LIN {X 0,Y 310.585,Z 527.407,A -85,B 0,C 180,E1 -15760.43,E2 -15760.43} C_VEL
LIN {X 0,Y 310.715,Z 527.488,A -85,B 0,C 180,E1 -15761.746,E2 -15761.746} C_VEL
LIN {X 0,Y 310.944,Z 526.948,A -85,B 0,C 180,E1 -15763.618,E2 -15763.618} C_VEL
LIN {X 0,Y 311.218,Z 525.347,A -85,B 0,C 180,E1 -15765.723,E2 -15765.723} C_VEL
LIN {X 0,Y 311.749,Z 522.836,A -85,B 0,C 180,E1 -15767.719,E2 -15767.719} C_VEL
LIN {X 0,Y 312.493,Z 519.275,A -85,B 0,C 180,E1 -15769.716,E2 -15769.716} C_VEL
LIN {X 0,Y 313.497,Z 514.55,A -85,B 0,C 180,E1 -15771.71,E2 -15771.71} C_VEL
LIN {X 0,Y 314.758,Z 508.405,A -85,B 0,C 180,E1 -15773.73,E2 -15773.73} C_VEL
LIN {X 0,Y 316.283,Z 500.927,A -85,B 0,C 180,E1 -15775.678,E2 -15775.678} C_VEL
LIN {X 0,Y 317.858,Z 493.142,A -85,B 0,C 180,E1 -15777.309,E2 -15777.309} C_VEL
LIN {X 0,Y 319.637,Z 483.592,A -85,B 0,C 180,E1 -15778.929,E2 -15778.929} C_VEL
LIN {X 0,Y 321.405,Z 472.884,A -85,B 0,C 180,E1 -15780.376,E2 -15780.376} C_VEL
LIN {X 0,Y 322.865,Z 462.517,A -85,B 0,C 180,E1 -15781.495,E2 -15781.495} C_VEL
LIN {X 0,Y 324.159,Z 451.225,A -85,B 0,C 180,E1 -15782.457,E2 -15782.457} C_VEL
LIN {X 0,Y 325.243,Z 438.611,A -85,B 0,C 180,E1 -15783.252,E2 -15783.252} C_VEL
LIN {X 0,Y 325.852,Z 426.556,A -85,B 0,C 180,E1 -15783.783,E2 -15783.783} C_VEL
LIN {X 0,Y 326.612,Z 407.281,A -85,B 0,C 180,E1 -15784.25,E2 -15784.25} C_VEL
LIN {X 0,Y 328.373,Z 349.267,A -85,B 0,C 180,E1 -15785.509,E2 -15785.509} C_VEL
LIN {X 0,Y 326.303,Z 343.527,A -85,B 0,C 180,E1 -15785.856,E2 -15785.856} C_VEL
LIN {X 0,Y 318.976,Z 327.276,A -85,B 0,C 180,E1 -15787.031,E2 -15787.031} C_VEL
LIN {X 0,Y 315.882,Z 321.035,A -85,B 0,C 180,E1 -15787.532,E2 -15787.532} C_VEL
LIN {X 0,Y 314.268,Z 318.796,A -85,B 0,C 180,E1 -15787.811,E2 -15787.811} C_VEL
LIN {X 0,Y 311.353,Z 316.882,A -85,B 0,C 180,E1 -15788.356,E2 -15788.356} C_VEL
LIN {X 0,Y 308.133,Z 315.361,A -85,B 0,C 180,E1 -15789.123,E2 -15789.123} C_VEL
LIN {X 0,Y 306.033,Z 313.784,A -85,B 0,C 180,E1 -15789.924,E2 -15789.924} C_VEL
LIN {X 0,Y 305.457,Z 312.436,A -85,B 0,C 180,E1 -15790.569,E2 -15790.569} C_VEL
LIN {X 0,Y 305.425,Z 312.439,A -85,B 0,C 180,E1 -15793.655,E2 -15793.655} C_VEL
LIN {X 0,Y 305.454,Z 312.435,A -85,B 0,C 180,E1 -15797.414,E2 -15797.414} C_VEL
LIN {X 0,Y 305.467,Z 312.429,A -85,B 0,C 180,E1 -15801.596,E2 -15801.596} C_VEL
LIN {X 0,Y 305.462,Z 312.43,A -85,B 0,C 180,E1 -15804.887,E2 -15804.887} C_VEL
LIN {X 0,Y 305.451,Z 312.427,A -85,B 0,C 180,E1 -15808.355,E2 -15808.355} C_VEL
LIN {X 0,Y 305.52,Z 312.423,A -85,B 0,C 180,E1 -15811.114,E2 -15811.114} C_VEL
LIN {X 0,Y 305.571,Z 312.415,A -85,B 0,C 180,E1 -15814.088,E2 -15814.088} C_VEL
LIN {X 0,Y 305.482,Z 312.428,A -85,B 0,C 180,E1 -15818.402,E2 -15818.402} C_VEL
LIN {X 0,Y 305.58,Z 312.412,A -85,B 0,C 180,E1 -15821.217,E2 -15821.217} C_VEL
LIN {X 0,Y 305.649,Z 312.404,A -85,B 0,C 180,E1 -15825.349,E2 -15825.349} C_VEL
LIN {X 0,Y 305.639,Z 312.405,A -85,B 0,C 180,E1 -15829.4,E2 -15829.4} C_VEL
LIN {X 0,Y 305.813,Z 312.388,A -85,B 0,C 180,E1 -15832.075,E2 -15832.075} C_VEL
LIN {X 0,Y 305.688,Z 312.403,A -85,B 0,C 180,E1 -15834.724,E2 -15834.724} C_VEL
LIN {X 0,Y 305.955,Z 312.367,A -85,B 0,C 180,E1 -15838.684,E2 -15838.684} C_VEL
LIN {X 0,Y 305.955,Z 312.37,A -85,B 0,C 180,E1 -15841.317,E2 -15841.317} C_VEL
LIN {X 0,Y 305.852,Z 312.375,A -85,B 0,C 180,E1 -15846.598,E2 -15846.598} C_VEL
LIN {X 0,Y 305.737,Z 312.397,A -85,B 0,C 180,E1 -15849.26,E2 -15849.26} C_VEL
LIN {X 0,Y 305.589,Z 312.415,A -85,B 0,C 180,E1 -15853.296,E2 -15853.296} C_VEL
LIN {X 0,Y 305.595,Z 312.409,A -85,B 0,C 180,E1 -15856.02,E2 -15856.02} C_VEL
LIN {X 0,Y 305.577,Z 312.415,A -85,B 0,C 180,E1 -15859.445,E2 -15859.445} C_VEL
LIN {X 0,Y 305.487,Z 312.43,A -85,B 0,C 180,E1 -15863.04,E2 -15863.04} C_VEL
LIN {X 0,Y 305.555,Z 312.422,A -85,B 0,C 180,E1 -15866.23,E2 -15866.23} C_VEL
LIN {X 0,Y 305.496,Z 312.425,A -85,B 0,C 180,E1 -15869.05,E2 -15869.05} C_VEL
LIN {X 0,Y 305.445,Z 312.431,A -85,B 0,C 180,E1 -15871.952,E2 -15871.952} C_VEL
LIN {X 0,Y 305.463,Z 312.431,A -85,B 0,C 180,E1 -15875.113,E2 -15875.113} C_VEL
LIN {X 0,Y 305.451,Z 312.432,A -85,B 0,C 180,E1 -15878.529,E2 -15878.529} C_VEL
LIN {X 0,Y 305.456,Z 312.433,A -85,B 0,C 180,E1 -15882.586,E2 -15882.586} C_VEL
LIN {X 0,Y 305.427,Z 312.438,A -85,B 0,C 180,E1 -15886.345,E2 -15886.345} C_VEL
LIN {X 0,Y 305.46,Z 312.437,A -85,B 0,C 180,E1 -15889.892,E2 -15889.892} C_VEL
LIN {X 0,Y 305.527,Z 312.594,A -85,B 0,C 180,E1 -15893.919,E2 -15893.919} C_VEL
LIN {X 0,Y 308.182,Z 323.12,A -85,B 0,C 180,E1 -15897.541,E2 -15897.541} C_VEL
LIN {X 0,Y 310.562,Z 333.507,A -85,B 0,C 180,E1 -15900.886,E2 -15900.886} C_VEL
LIN {X 0,Y 311.27,Z 336.978,A -85,B 0,C 180,E1 -15901.907,E2 -15901.907} C_VEL
LIN {X 0,Y 314.189,Z 344.264,A -85,B 0,C 180,E1 -15902.425,E2 -15902.425} C_VEL
LIN {X 0,Y 319.342,Z 369.476,A -85,B 0,C 180,E1 -15903.626,E2 -15903.626} C_VEL
LIN {X 0,Y 321.296,Z 381.976,A -85,B 0,C 180,E1 -15904.142,E2 -15904.142} C_VEL
LIN {X 0,Y 319.435,Z 445.643,A -85,B 0,C 180,E1 -15905.593,E2 -15905.593} C_VEL
LIN {X 0,Y 318.464,Z 458.812,A -85,B 0,C 180,E1 -15906.12,E2 -15906.12} C_VEL
LIN {X 0,Y 317.004,Z 472.041,A -85,B 0,C 180,E1 -15906.912,E2 -15906.912} C_VEL
LIN {X 0,Y 315.443,Z 483.946,A -85,B 0,C 180,E1 -15907.915,E2 -15907.915} C_VEL
LIN {X 0,Y 313.482,Z 495.373,A -85,B 0,C 180,E1 -15909.151,E2 -15909.151} C_VEL
LIN {X 0,Y 311.609,Z 505.685,A -85,B 0,C 180,E1 -15910.569,E2 -15910.569} C_VEL
LIN {X 0,Y 309.728,Z 514.983,A -85,B 0,C 180,E1 -15912.162,E2 -15912.162} C_VEL
LIN {X 0,Y 308.021,Z 523.994,A -85,B 0,C 180,E1 -15914.109,E2 -15914.109} C_VEL
LIN {X 0,Y 306.542,Z 531.283,A -85,B 0,C 180,E1 -15916.07,E2 -15916.07} C_VEL
LIN {X 0,Y 305.289,Z 537.146,A -85,B 0,C 180,E1 -15918.042,E2 -15918.042} C_VEL
LIN {X 0,Y 304.495,Z 541.787,A -85,B 0,C 180,E1 -15920.031,E2 -15920.031} C_VEL
LIN {X 0,Y 303.991,Z 545.34,A -85,B 0,C 180,E1 -15922.026,E2 -15922.026} C_VEL
LIN {X 0,Y 303.661,Z 548.289,A -85,B 0,C 180,E1 -15924.388,E2 -15924.388} C_VEL
LIN {X 0,Y 303.633,Z 549.542,A -85,B 0,C 180,E1 -15926.018,E2 -15926.018} C_VEL
LIN {X 0,Y 303.624,Z 550.149,A -85,B 0,C 180,E1 -15927.346,E2 -15927.346} C_VEL
LIN {X 0,Y 303.608,Z 550.349,A -85,B 0,C 180,E1 -15928.673,E2 -15928.673} C_VEL
LIN {X 0,Y 303.669,Z 550.127,A -85,B 0,C 180,E1 -15930,E2 -15930} C_VEL
LIN {X 0,Y 303.635,Z 549.511,A -85,B 0,C 180,E1 -15931.326,E2 -15931.326} C_VEL
LIN {X 0,Y 303.646,Z 548.504,A -85,B 0,C 180,E1 -15932.653,E2 -15932.653} C_VEL
LIN {X 0,Y 303.671,Z 547.075,A -85,B 0,C 180,E1 -15933.981,E2 -15933.981} C_VEL
LIN {X 0,Y 303.684,Z 544.618,A -85,B 0,C 180,E1 -15935.655,E2 -15935.655} C_VEL
LIN {X 0,Y 303.939,Z 540.041,A -85,B 0,C 180,E1 -15937.974,E2 -15937.974} C_VEL
LIN {X 0,Y 304.438,Z 533.793,A -85,B 0,C 180,E1 -15940.306,E2 -15940.306} C_VEL
LIN {X 0,Y 305.137,Z 526.972,A -85,B 0,C 180,E1 -15942.3,E2 -15942.3} C_VEL
LIN {X 0,Y 306.181,Z 518.49,A -85,B 0,C 180,E1 -15944.285,E2 -15944.285} C_VEL
LIN {X 0,Y 307.33,Z 509.737,A -85,B 0,C 180,E1 -15945.927,E2 -15945.927} C_VEL
LIN {X 0,Y 308.489,Z 498.922,A -85,B 0,C 180,E1 -15947.569,E2 -15947.569} C_VEL
LIN {X 0,Y 309.773,Z 488.174,A -85,B 0,C 180,E1 -15948.862,E2 -15948.862} C_VEL
LIN {X 0,Y 311.023,Z 476.109,A -85,B 0,C 180,E1 -15949.984,E2 -15949.984} C_VEL
LIN {X 0,Y 312.081,Z 463.518,A -85,B 0,C 180,E1 -15950.86,E2 -15950.86} C_VEL
LIN {X 0,Y 312.989,Z 450.349,A -85,B 0,C 180,E1 -15951.486,E2 -15951.486} C_VEL
LIN {X 0,Y 313.357,Z 436.065,A -85,B 0,C 180,E1 -15951.892,E2 -15951.892} C_VEL
LIN {X 0,Y 314.514,Z 379.407,A -85,B 0,C 180,E1 -15953.167,E2 -15953.167} C_VEL
LIN {X 0,Y 308.841,Z 337.463,A -85,B 0,C 180,E1 -15954.577,E2 -15954.577} C_VEL
LIN {X 0,Y 309.378,Z 332.279,A -85,B 0,C 180,E1 -15955.931,E2 -15955.931} C_VEL
LIN {X 0,Y 307.949,Z 323.986,A -85,B 0,C 180,E1 -15958.28,E2 -15958.28} C_VEL
LIN {X 0,Y 305.465,Z 312.438,A -85,B 0,C 180,E1 -15961.706,E2 -15961.706} C_VEL
LIN {X 0,Y 305.462,Z 312.433,A -85,B 0,C 180,E1 -15965.112,E2 -15965.112} C_VEL
LIN {X 0,Y 305.466,Z 312.436,A -85,B 0,C 180,E1 -15968.532,E2 -15968.532} C_VEL
LIN {X 0,Y 305.453,Z 312.438,A -85,B 0,C 180,E1 -15972.585,E2 -15972.585} C_VEL
LIN {X 0,Y 305.423,Z 312.441,A -85,B 0,C 180,E1 -15976.344,E2 -15976.344} C_VEL
LIN {X 0,Y 305.456,Z 312.434,A -85,B 0,C 180,E1 -15979.892,E2 -15979.892} C_VEL
LIN {X 0,Y 305.478,Z 312.431,A -85,B 0,C 180,E1 -15983.631,E2 -15983.631} C_VEL
LIN {X 0,Y 305.462,Z 312.436,A -85,B 0,C 180,E1 -15986.483,E2 -15986.483} C_VEL
LIN {X 0,Y 305.455,Z 312.435,A -85,B 0,C 180,E1 -15989.59,E2 -15989.59} C_VEL
LIN {X 0,Y 305.511,Z 312.429,A -85,B 0,C 180,E1 -15992.607,E2 -15992.607} C_VEL
LIN {X 0,Y 305.505,Z 312.429,A -85,B 0,C 180,E1 -15995.538,E2 -15995.538} C_VEL
LIN {X 0,Y 305.516,Z 312.426,A -85,B 0,C 180,E1 -15999.814,E2 -15999.814} C_VEL
LIN {X 0,Y 305.571,Z 312.419,A -85,B 0,C 180,E1 -16002.602,E2 -16002.602} C_VEL
LIN {X 0,Y 305.645,Z 312.413,A -85,B 0,C 180,E1 -16005.348,E2 -16005.348} C_VEL
LIN {X 0,Y 305.634,Z 312.409,A -85,B 0,C 180,E1 -16009.399,E2 -16009.399} C_VEL
LIN {X 0,Y 305.804,Z 312.39,A -85,B 0,C 180,E1 -16012.074,E2 -16012.074} C_VEL
LIN {X 0,Y 305.682,Z 312.405,A -85,B 0,C 180,E1 -16014.723,E2 -16014.723} C_VEL
LIN {X 0,Y 305.952,Z 312.365,A -85,B 0,C 180,E1 -16018.683,E2 -16018.683} C_VEL
LIN {X 0,Y 305.951,Z 312.369,A -85,B 0,C 180,E1 -16021.316,E2 -16021.316} C_VEL
LIN {X 0,Y 305.671,Z 312.407,A -85,B 0,C 180,E1 -16025.277,E2 -16025.277} C_VEL
LIN {X 0,Y 305.76,Z 312.396,A -85,B 0,C 180,E1 -16027.927,E2 -16027.927} C_VEL
LIN {X 0,Y 305.599,Z 312.416,A -85,B 0,C 180,E1 -16031.945,E2 -16031.945} C_VEL
LIN {X 0,Y 305.633,Z 312.411,A -85,B 0,C 180,E1 -16035.035,E2 -16035.035} C_VEL
LIN {X 0,Y 305.575,Z 312.415,A -85,B 0,C 180,E1 -16038.783,E2 -16038.783} C_VEL
LIN {X 0,Y 305.481,Z 312.429,A -85,B 0,C 180,E1 -16043.039,E2 -16043.039} C_VEL
LIN {X 0,Y 305.543,Z 312.426,A -85,B 0,C 180,E1 -16046.227,E2 -16046.227} C_VEL
LIN {X 0,Y 305.491,Z 312.425,A -85,B 0,C 180,E1 -16049.05,E2 -16049.05} C_VEL
LIN {X 0,Y 305.46,Z 312.432,A -85,B 0,C 180,E1 -16053.517,E2 -16053.517} C_VEL
LIN {X 0,Y 305.468,Z 312.434,A -85,B 0,C 180,E1 -16056.74,E2 -16056.74} C_VEL
LIN {X 0,Y 305.45,Z 312.434,A -85,B 0,C 180,E1 -16060.6,E2 -16060.6} C_VEL
LIN {X 0,Y 305.421,Z 312.437,A -85,B 0,C 180,E1 -16063.656,E2 -16063.656} C_VEL
LIN {X 0,Y 305.431,Z 312.438,A -85,B 0,C 180,E1 -16067.419,E2 -16067.419} C_VEL
LIN {X 0,Y 305.456,Z 312.433,A -85,B 0,C 180,E1 -16071.596,E2 -16071.596} C_VEL
LIN {X 0,Y 305.458,Z 312.435,A -85,B 0,C 180,E1 -16074.887,E2 -16074.887} C_VEL
LIN {X 0,Y 305.438,Z 312.435,A -85,B 0,C 180,E1 -16078.359,E2 -16078.359} C_VEL
LIN {X 0,Y 305.461,Z 312.434,A -85,B 0,C 180,E1 -16081.109,E2 -16081.109} C_VEL
LIN {X 0,Y 305.476,Z 312.431,A -85,B 0,C 180,E1 -16084.08,E2 -16084.08} C_VEL
LIN {X 0,Y 305.471,Z 312.432,A -85,B 0,C 180,E1 -16088.401,E2 -16088.401} C_VEL
LIN {X 0,Y 305.541,Z 312.425,A -85,B 0,C 180,E1 -16091.215,E2 -16091.215} C_VEL
LIN {X 0,Y 305.601,Z 312.487,A -85,B 0,C 180,E1 -16094.041,E2 -16094.041} C_VEL
LIN {X 0,Y 306.551,Z 316.889,A -85,B 0,C 180,E1 -16095.359,E2 -16095.359} C_VEL
LIN {X 0,Y 313.107,Z 335.617,A -85,B 0,C 180,E1 -16096.279,E2 -16096.279} C_VEL
LIN {X 0,Y 314.384,Z 341.929,A -85,B 0,C 180,E1 -16096.518,E2 -16096.518} C_VEL
LIN {X 0,Y 315.143,Z 347.62,A -85,B 0,C 180,E1 -16096.704,E2 -16096.704} C_VEL
LIN {X 0,Y 313.441,Z 423.804,A -85,B 0,C 180,E1 -16098.44,E2 -16098.44} C_VEL
LIN {X 0,Y 312.86,Z 437.018,A -85,B 0,C 180,E1 -16098.993,E2 -16098.993} C_VEL
LIN {X 0,Y 312.115,Z 449.671,A -85,B 0,C 180,E1 -16099.787,E2 -16099.787} C_VEL
LIN {X 0,Y 311.196,Z 460.961,A -85,B 0,C 180,E1 -16100.741,E2 -16100.741} C_VEL
LIN {X 0,Y 310.227,Z 468.585,A -85,B 0,C 180,E1 -16101.533,E2 -16101.533} C_VEL
LIN {X 0,Y 309.04,Z 478.731,A -85,B 0,C 180,E1 -16102.815,E2 -16102.815} C_VEL
LIN {X 0,Y 307.809,Z 488.97,A -85,B 0,C 180,E1 -16104.432,E2 -16104.432} C_VEL
LIN {X 0,Y 306.798,Z 497.282,A -85,B 0,C 180,E1 -16106.06,E2 -16106.06} C_VEL
LIN {X 0,Y 305.735,Z 505.425,A -85,B 0,C 180,E1 -16108.024,E2 -16108.024} C_VEL
LIN {X 0,Y 304.91,Z 511.985,A -85,B 0,C 180,E1 -16110,E2 -16110} C_VEL
LIN {X 0,Y 304.405,Z 517.207,A -85,B 0,C 180,E1 -16111.985,E2 -16111.985} C_VEL
LIN {X 0,Y 304.021,Z 521.279,A -85,B 0,C 180,E1 -16113.977,E2 -16113.977} C_VEL
LIN {X 0,Y 303.924,Z 524.465,A -85,B 0,C 180,E1 -16116.1,E2 -16116.1} C_VEL
LIN {X 0,Y 303.626,Z 526.365,A -85,B 0,C 180,E1 -16117.984,E2 -16117.984} C_VEL
LIN {X 0,Y 303.519,Z 527.251,A -85,B 0,C 180,E1 -16119.328,E2 -16119.328} C_VEL
LIN {X 0,Y 303.64,Z 527.738,A -85,B 0,C 180,E1 -16122.024,E2 -16122.024} C_VEL
LIN {X 0,Y 303.86,Z 527.246,A -85,B 0,C 180,E1 -16123.732,E2 -16123.732} C_VEL
LIN {X 0,Y 304.208,Z 525.448,A -85,B 0,C 180,E1 -16126.095,E2 -16126.095} C_VEL
LIN {X 0,Y 304.814,Z 522.858,A -85,B 0,C 180,E1 -16128.136,E2 -16128.136} C_VEL
LIN {X 0,Y 305.62,Z 519.213,A -85,B 0,C 180,E1 -16130.178,E2 -16130.178} C_VEL
LIN {X 0,Y 306.697,Z 514.397,A -85,B 0,C 180,E1 -16132.216,E2 -16132.216} C_VEL
LIN {X 0,Y 308.046,Z 508.257,A -85,B 0,C 180,E1 -16134.247,E2 -16134.247} C_VEL
LIN {X 0,Y 309.726,Z 500.565,A -85,B 0,C 180,E1 -16136.262,E2 -16136.262} C_VEL
LIN {X 0,Y 311.379,Z 492.632,A -85,B 0,C 180,E1 -16137.927,E2 -16137.927} C_VEL
LIN {X 0,Y 313.251,Z 482.861,A -85,B 0,C 180,E1 -16139.577,E2 -16139.577} C_VEL
LIN {X 0,Y 315.13,Z 471.947,A -85,B 0,C 180,E1 -16141.047,E2 -16141.047} C_VEL
LIN {X 0,Y 316.664,Z 461.296,A -85,B 0,C 180,E1 -16142.185,E2 -16142.185} C_VEL
LIN {X 0,Y 317.945,Z 450.263,A -85,B 0,C 180,E1 -16143.106,E2 -16143.106} C_VEL
LIN {X 0,Y 319,Z 437.583,A -85,B 0,C 180,E1 -16143.895,E2 -16143.895} C_VEL
LIN {X 0,Y 319.622,Z 426.086,A -85,B 0,C 180,E1 -16144.391,E2 -16144.391} C_VEL
LIN {X 0,Y 320.592,Z 400.835,A -85,B 0,C 180,E1 -16144.988,E2 -16144.988} C_VEL
LIN {X 0,Y 322.138,Z 350.538,A -85,B 0,C 180,E1 -16146.103,E2 -16146.103} C_VEL
LIN {X 0,Y 314.896,Z 333.66,A -85,B 0,C 180,E1 -16147.31,E2 -16147.31} C_VEL
LIN {X 0,Y 306.704,Z 317.207,A -85,B 0,C 180,E1 -16148.722,E2 -16148.722} C_VEL
LIN {X 0,Y 305.465,Z 312.435,A -85,B 0,C 180,E1 -16150.489,E2 -16150.489} C_VEL
LIN {X 0,Y 305.457,Z 312.436,A -85,B 0,C 180,E1 -16150.569,E2 -16150.569} C_VEL
LIN {X 0,Y 304.712,Z 312.532,A -85,B 0,C 180,E1 -16151.667,E2 -16151.667} C_VEL
LIN {X 0,Y 301.799,Z 312.892,A -85,B 0,C 180,E1 -16153.455,E2 -16153.455} C_VEL
LIN {X 0,Y 299.399,Z 313.189,A -85,B 0,C 180,E1 -16154.906,E2 -16154.906} C_VEL
LIN {X 0,Y 298.415,Z 313.313,A -85,B 0,C 180,E1 -16156.029,E2 -16156.029} C_VEL
LIN {X 0,Y 298.356,Z 313.317,A -85,B 0,C 180,E1 -16156.41,E2 -16156.41} C_VEL
LIN {X 0,Y 298.4,Z 313.312,A -85,B 0,C 180,E1 -16160.513,E2 -16160.513} C_VEL
LIN {X 0,Y 298.417,Z 313.307,A -85,B 0,C 180,E1 -16163.93,E2 -16163.93} C_VEL
LIN {X 0,Y 298.395,Z 313.307,A -85,B 0,C 180,E1 -16167.984,E2 -16167.984} C_VEL
LIN {X 0,Y 298.463,Z 313.296,A -85,B 0,C 180,E1 -16171.905,E2 -16171.905} C_VEL
LIN {X 0,Y 298.484,Z 313.3,A -85,B 0,C 180,E1 -16174.924,E2 -16174.924} C_VEL
LIN {X 0,Y 298.437,Z 313.306,A -85,B 0,C 180,E1 -16179.315,E2 -16179.315} C_VEL
LIN {X 0,Y 298.535,Z 313.297,A -85,B 0,C 180,E1 -16182.179,E2 -16182.179} C_VEL
LIN {X 0,Y 298.593,Z 313.281,A -85,B 0,C 180,E1 -16184.995,E2 -16184.995} C_VEL
LIN {X 0,Y 298.594,Z 313.282,A -85,B 0,C 180,E1 -16189.147,E2 -16189.147} C_VEL
LIN {X 0,Y 298.759,Z 313.269,A -85,B 0,C 180,E1 -16191.886,E2 -16191.886} C_VEL
LIN {X 0,Y 298.659,Z 313.279,A -85,B 0,C 180,E1 -16194.599,E2 -16194.599} C_VEL
LIN {X 0,Y 298.922,Z 313.242,A -85,B 0,C 180,E1 -16198.653,E2 -16198.653} C_VEL
LIN {X 0,Y 298.922,Z 313.246,A -85,B 0,C 180,E1 -16201.348,E2 -16201.348} C_VEL
LIN {X 0,Y 298.797,Z 313.252,A -85,B 0,C 180,E1 -16206.754,E2 -16206.754} C_VEL
LIN {X 0,Y 298.681,Z 313.276,A -85,B 0,C 180,E1 -16209.481,E2 -16209.481} C_VEL
LIN {X 0,Y 298.553,Z 313.292,A -85,B 0,C 180,E1 -16213.616,E2 -16213.616} C_VEL
LIN {X 0,Y 298.55,Z 313.286,A -85,B 0,C 180,E1 -16216.409,E2 -16216.409} C_VEL
LIN {X 0,Y 298.511,Z 313.295,A -85,B 0,C 180,E1 -16219.654,E2 -16219.654} C_VEL
LIN {X 0,Y 298.43,Z 313.307,A -85,B 0,C 180,E1 -16223.6,E2 -16223.6} C_VEL
LIN {X 0,Y 298.493,Z 313.304,A -85,B 0,C 180,E1 -16226.574,E2 -16226.574} C_VEL
LIN {X 0,Y 298.422,Z 313.311,A -85,B 0,C 180,E1 -16229.641,E2 -16229.641} C_VEL
LIN {X 0,Y 298.397,Z 313.309,A -85,B 0,C 180,E1 -16232.8,E2 -16232.8} C_VEL
LIN {X 0,Y 298.448,Z 313.304,A -85,B 0,C 180,E1 -16236.808,E2 -16236.808} C_VEL
LIN {X 0,Y 298.388,Z 313.293,A -85,B 0,C 180,E1 -16241.088,E2 -16241.088} C_VEL
LIN {X 0,Y 298.4,Z 313.315,A -85,B 0,C 180,E1 -16243.103,E2 -16243.103} C_VEL
LIN {X 0,Y 298.405,Z 313.312,A -85,B 0,C 180,E1 -16246.921,E2 -16246.921} C_VEL
LIN {X 0,Y 298.406,Z 313.314,A -85,B 0,C 180,E1 -16251.006,E2 -16251.006} C_VEL
LIN {X 0,Y 298.467,Z 313.503,A -85,B 0,C 180,E1 -16253.188,E2 -16253.188} C_VEL
LIN {X 0,Y 300.93,Z 323.149,A -85,B 0,C 180,E1 -16256.634,E2 -16256.634} C_VEL
LIN {X 0,Y 303.403,Z 333.599,A -85,B 0,C 180,E1 -16260.13,E2 -16260.13} C_VEL
LIN {X 0,Y 304.041,Z 336.64,A -85,B 0,C 180,E1 -16261.054,E2 -16261.054} C_VEL
LIN {X 0,Y 308.401,Z 346.881,A -85,B 0,C 180,E1 -16261.846,E2 -16261.846} C_VEL
LIN {X 0,Y 313.301,Z 371.316,A -85,B 0,C 180,E1 -16263.038,E2 -16263.038} C_VEL
LIN {X 0,Y 315.086,Z 383.682,A -85,B 0,C 180,E1 -16263.549,E2 -16263.549} C_VEL
LIN {X 0,Y 313.182,Z 445.468,A -85,B 0,C 180,E1 -16264.984,E2 -16264.984} C_VEL
LIN {X 0,Y 312.177,Z 458.601,A -85,B 0,C 180,E1 -16265.52,E2 -16265.52} C_VEL
LIN {X 0,Y 310.659,Z 471.811,A -85,B 0,C 180,E1 -16266.324,E2 -16266.324} C_VEL
LIN {X 0,Y 309.113,Z 482.919,A -85,B 0,C 180,E1 -16267.262,E2 -16267.262} C_VEL
LIN {X 0,Y 307.144,Z 494.476,A -85,B 0,C 180,E1 -16268.524,E2 -16268.524} C_VEL
LIN {X 0,Y 305.124,Z 504.895,A -85,B 0,C 180,E1 -16269.963,E2 -16269.963} C_VEL
LIN {X 0,Y 303.355,Z 513.431,A -85,B 0,C 180,E1 -16271.424,E2 -16271.424} C_VEL
LIN {X 0,Y 301.598,Z 521.885,A -85,B 0,C 180,E1 -16273.2,E2 -16273.2} C_VEL
LIN {X 0,Y 300.164,Z 529.064,A -85,B 0,C 180,E1 -16275.075,E2 -16275.075} C_VEL
LIN {X 0,Y 298.695,Z 535.293,A -85,B 0,C 180,E1 -16277.083,E2 -16277.083} C_VEL
LIN {X 0,Y 297.736,Z 540.268,A -85,B 0,C 180,E1 -16279.115,E2 -16279.115} C_VEL
LIN {X 0,Y 297.09,Z 544.133,A -85,B 0,C 180,E1 -16281.154,E2 -16281.154} C_VEL
LIN {X 0,Y 296.691,Z 546.99,A -85,B 0,C 180,E1 -16283.198,E2 -16283.198} C_VEL
LIN {X 0,Y 296.531,Z 549.326,A -85,B 0,C 180,E1 -16285.922,E2 -16285.922} C_VEL
LIN {X 0,Y 296.549,Z 549.914,A -85,B 0,C 180,E1 -16287.283,E2 -16287.283} C_VEL
LIN {X 0,Y 296.525,Z 550.075,A -85,B 0,C 180,E1 -16288.641,E2 -16288.641} C_VEL
LIN {X 0,Y 296.581,Z 549.832,A -85,B 0,C 180,E1 -16290,E2 -16290} C_VEL
LIN {X 0,Y 296.551,Z 549.196,A -85,B 0,C 180,E1 -16291.357,E2 -16291.357} C_VEL
LIN {X 0,Y 296.571,Z 548.169,A -85,B 0,C 180,E1 -16292.716,E2 -16292.716} C_VEL
LIN {X 0,Y 296.587,Z 546.699,A -85,B 0,C 180,E1 -16294.076,E2 -16294.076} C_VEL
LIN {X 0,Y 296.638,Z 543.675,A -85,B 0,C 180,E1 -16296.119,E2 -16296.119} C_VEL
LIN {X 0,Y 296.873,Z 539.576,A -85,B 0,C 180,E1 -16298.165,E2 -16298.165} C_VEL
LIN {X 0,Y 297.408,Z 533.268,A -85,B 0,C 180,E1 -16300.552,E2 -16300.552} C_VEL
LIN {X 0,Y 298.175,Z 526.392,A -85,B 0,C 180,E1 -16302.592,E2 -16302.592} C_VEL
LIN {X 0,Y 299.082,Z 519.371,A -85,B 0,C 180,E1 -16304.284,E2 -16304.284} C_VEL
LIN {X 0,Y 300.225,Z 510.909,A -85,B 0,C 180,E1 -16305.965,E2 -16305.965} C_VEL
LIN {X 0,Y 301.34,Z 500.421,A -85,B 0,C 180,E1 -16307.649,E2 -16307.649} C_VEL
LIN {X 0,Y 302.615,Z 490.054,A -85,B 0,C 180,E1 -16308.973,E2 -16308.973} C_VEL
LIN {X 0,Y 303.945,Z 478.711,A -85,B 0,C 180,E1 -16310.117,E2 -16310.117} C_VEL
LIN {X 0,Y 305.02,Z 467.148,A -85,B 0,C 180,E1 -16311.012,E2 -16311.012} C_VEL
LIN {X 0,Y 306.024,Z 453.877,A -85,B 0,C 180,E1 -16311.735,E2 -16311.735} C_VEL
LIN {X 0,Y 306.565,Z 440.969,A -85,B 0,C 180,E1 -16312.181,E2 -16312.181} C_VEL
LIN {X 0,Y 307.811,Z 380.639,A -85,B 0,C 180,E1 -16313.575,E2 -16313.575} C_VEL
LIN {X 0,Y 302.735,Z 342.14,A -85,B 0,C 180,E1 -16314.878,E2 -16314.878} C_VEL
LIN {X 0,Y 302.007,Z 337.218,A -85,B 0,C 180,E1 -16315.068,E2 -16315.068} C_VEL
LIN {X 0,Y 302.386,Z 332.983,A -85,B 0,C 180,E1 -16316.205,E2 -16316.205} C_VEL
LIN {X 0,Y 300.593,Z 323.34,A -85,B 0,C 180,E1 -16319.021,E2 -16319.021} C_VEL
LIN {X 0,Y 298.407,Z 313.317,A -85,B 0,C 180,E1 -16322.12,E2 -16322.12} C_VEL
LIN {X 0,Y 298.418,Z 313.314,A -85,B 0,C 180,E1 -16326.069,E2 -16326.069} C_VEL
LIN {X 0,Y 298.408,Z 313.312,A -85,B 0,C 180,E1 -16329.485,E2 -16329.485} C_VEL
LIN {X 0,Y 298.397,Z 313.313,A -85,B 0,C 180,E1 -16333.102,E2 -16333.102} C_VEL
LIN {X 0,Y 298.401,Z 313.315,A -85,B 0,C 180,E1 -16336.92,E2 -16336.92} C_VEL
LIN {X 0,Y 298.396,Z 313.316,A -85,B 0,C 180,E1 -16341.007,E2 -16341.007} C_VEL
LIN {X 0,Y 298.415,Z 313.312,A -85,B 0,C 180,E1 -16343.929,E2 -16343.929} C_VEL
LIN {X 0,Y 298.39,Z 313.314,A -85,B 0,C 180,E1 -16347.983,E2 -16347.983} C_VEL
LIN {X 0,Y 298.454,Z 313.306,A -85,B 0,C 180,E1 -16351.903,E2 -16351.903} C_VEL
LIN {X 0,Y 298.48,Z 313.307,A -85,B 0,C 180,E1 -16354.923,E2 -16354.923} C_VEL
LIN {X 0,Y 298.447,Z 313.311,A -85,B 0,C 180,E1 -16359.315,E2 -16359.315} C_VEL
LIN {X 0,Y 298.534,Z 313.294,A -85,B 0,C 180,E1 -16362.179,E2 -16362.179} C_VEL
LIN {X 0,Y 298.59,Z 313.291,A -85,B 0,C 180,E1 -16364.994,E2 -16364.994} C_VEL
LIN {X 0,Y 298.589,Z 313.285,A -85,B 0,C 180,E1 -16369.146,E2 -16369.146} C_VEL
LIN {X 0,Y 298.751,Z 313.27,A -85,B 0,C 180,E1 -16371.885,E2 -16371.885} C_VEL
LIN {X 0,Y 298.653,Z 313.28,A -85,B 0,C 180,E1 -16374.598,E2 -16374.598} C_VEL
LIN {X 0,Y 298.919,Z 313.241,A -85,B 0,C 180,E1 -16378.652,E2 -16378.652} C_VEL
LIN {X 0,Y 298.917,Z 313.245,A -85,B 0,C 180,E1 -16381.347,E2 -16381.347} C_VEL
LIN {X 0,Y 298.64,Z 313.284,A -85,B 0,C 180,E1 -16385.401,E2 -16385.401} C_VEL
LIN {X 0,Y 298.708,Z 313.272,A -85,B 0,C 180,E1 -16388.115,E2 -16388.115} C_VEL
LIN {X 0,Y 298.549,Z 313.296,A -85,B 0,C 180,E1 -16392.231,E2 -16392.231} C_VEL
LIN {X 0,Y 298.601,Z 313.287,A -85,B 0,C 180,E1 -16395.209,E2 -16395.209} C_VEL
LIN {X 0,Y 298.52,Z 313.292,A -85,B 0,C 180,E1 -16399.244,E2 -16399.244} C_VEL
LIN {X 0,Y 298.424,Z 313.308,A -85,B 0,C 180,E1 -16403.6,E2 -16403.6} C_VEL
LIN {X 0,Y 298.485,Z 313.304,A -85,B 0,C 180,E1 -16406.575,E2 -16406.575} C_VEL
LIN {X 0,Y 298.416,Z 313.304,A -85,B 0,C 180,E1 -16409.641,E2 -16409.641} C_VEL
LIN {X 0,Y 298.391,Z 313.316,A -85,B 0,C 180,E1 -16412.8,E2 -16412.8} C_VEL
LIN {X 0,Y 298.44,Z 313.308,A -85,B 0,C 180,E1 -16416.807,E2 -16416.807} C_VEL
LIN {X 0,Y 298.383,Z 313.317,A -85,B 0,C 180,E1 -16421.088,E2 -16421.088} C_VEL
LIN {X 0,Y 298.395,Z 313.315,A -85,B 0,C 180,E1 -16423.104,E2 -16423.104} C_VEL
LIN {X 0,Y 298.367,Z 313.316,A -85,B 0,C 180,E1 -16426.915,E2 -16426.915} C_VEL
LIN {X 0,Y 298.381,Z 313.318,A -85,B 0,C 180,E1 -16431.011,E2 -16431.011} C_VEL
LIN {X 0,Y 298.413,Z 313.311,A -85,B 0,C 180,E1 -16433.93,E2 -16433.93} C_VEL
LIN {X 0,Y 298.389,Z 313.318,A -85,B 0,C 180,E1 -16437.2,E2 -16437.2} C_VEL
LIN {X 0,Y 298.367,Z 313.314,A -85,B 0,C 180,E1 -16440.636,E2 -16440.636} C_VEL
LIN {X 0,Y 298.419,Z 313.31,A -85,B 0,C 180,E1 -16444.919,E2 -16444.919} C_VEL
LIN {X 0,Y 298.405,Z 313.315,A -85,B 0,C 180,E1 -16447.863,E2 -16447.863} C_VEL
LIN {X 0,Y 298.501,Z 313.301,A -85,B 0,C 180,E1 -16450.755,E2 -16450.755} C_VEL
LIN {X 0,Y 298.535,Z 313.341,A -85,B 0,C 180,E1 -16453.662,E2 -16453.662} C_VEL
LIN {X 0,Y 299.396,Z 317.182,A -85,B 0,C 180,E1 -16454.834,E2 -16454.834} C_VEL
LIN {X 0,Y 306.101,Z 335.932,A -85,B 0,C 180,E1 -16455.798,E2 -16455.798} C_VEL
LIN {X 0,Y 307.468,Z 341.277,A -85,B 0,C 180,E1 -16456.027,E2 -16456.027} C_VEL
LIN {X 0,Y 308.476,Z 348.543,A -85,B 0,C 180,E1 -16456.275,E2 -16456.275} C_VEL
LIN {X 0,Y 306.678,Z 424.899,A -85,B 0,C 180,E1 -16458.061,E2 -16458.061} C_VEL
LIN {X 0,Y 306.053,Z 438.5,A -85,B 0,C 180,E1 -16458.661,E2 -16458.661} C_VEL
LIN {X 0,Y 305.27,Z 450.829,A -85,B 0,C 180,E1 -16459.471,E2 -16459.471} C_VEL
LIN {X 0,Y 304.262,Z 462.651,A -85,B 0,C 180,E1 -16460.528,E2 -16460.528} C_VEL
LIN {X 0,Y 302.715,Z 474.078,A -85,B 0,C 180,E1 -16461.825,E2 -16461.825} C_VEL
LIN {X 0,Y 301.559,Z 484.304,A -85,B 0,C 180,E1 -16463.309,E2 -16463.309} C_VEL
LIN {X 0,Y 300.305,Z 493.515,A -85,B 0,C 180,E1 -16464.966,E2 -16464.966} C_VEL
LIN {X 0,Y 299.188,Z 502.442,A -85,B 0,C 180,E1 -16466.971,E2 -16466.971} C_VEL
LIN {X 0,Y 298.188,Z 509.655,A -85,B 0,C 180,E1 -16468.988,E2 -16468.988} C_VEL
LIN {X 0,Y 297.661,Z 514.517,A -85,B 0,C 180,E1 -16470.677,E2 -16470.677} C_VEL
LIN {X 0,Y 297.088,Z 519.259,A -85,B 0,C 180,E1 -16472.712,E2 -16472.712} C_VEL
LIN {X 0,Y 296.899,Z 522.883,A -85,B 0,C 180,E1 -16474.753,E2 -16474.753} C_VEL
LIN {X 0,Y 296.699,Z 525.511,A -85,B 0,C 180,E1 -16476.802,E2 -16476.802} C_VEL
LIN {X 0,Y 296.509,Z 526.76,A -85,B 0,C 180,E1 -16478.176,E2 -16478.176} C_VEL
LIN {X 0,Y 296.428,Z 527.58,A -85,B 0,C 180,E1 -16479.554,E2 -16479.554} C_VEL
LIN {X 0,Y 296.573,Z 527.987,A -85,B 0,C 180,E1 -16482.315,E2 -16482.315} C_VEL
LIN {X 0,Y 296.782,Z 527.54,A -85,B 0,C 180,E1 -16483.855,E2 -16483.855} C_VEL
LIN {X 0,Y 297.234,Z 525.548,A -85,B 0,C 180,E1 -16486.484,E2 -16486.484} C_VEL
LIN {X 0,Y 297.888,Z 522.881,A -85,B 0,C 180,E1 -16488.573,E2 -16488.573} C_VEL
LIN {X 0,Y 298.768,Z 519.151,A -85,B 0,C 180,E1 -16490.662,E2 -16490.662} C_VEL
LIN {X 0,Y 299.958,Z 514.246,A -85,B 0,C 180,E1 -16492.743,E2 -16492.743} C_VEL
LIN {X 0,Y 301.357,Z 508.005,A -85,B 0,C 180,E1 -16494.821,E2 -16494.821} C_VEL
LIN {X 0,Y 303.179,Z 500.167,A -85,B 0,C 180,E1 -16496.874,E2 -16496.874} C_VEL
LIN {X 0,Y 304.917,Z 492.073,A -85,B 0,C 180,E1 -16498.572,E2 -16498.572} C_VEL
LIN {X 0,Y 306.944,Z 482.143,A -85,B 0,C 180,E1 -16500.247,E2 -16500.247} C_VEL
LIN {X 0,Y 308.664,Z 472.347,A -85,B 0,C 180,E1 -16501.58,E2 -16501.58} C_VEL
LIN {X 0,Y 310.268,Z 461.74,A -85,B 0,C 180,E1 -16502.738,E2 -16502.738} C_VEL
LIN {X 0,Y 311.687,Z 449.946,A -85,B 0,C 180,E1 -16503.734,E2 -16503.734} C_VEL
LIN {X 0,Y 312.77,Z 437.413,A -85,B 0,C 180,E1 -16504.519,E2 -16504.519} C_VEL
LIN {X 0,Y 313.419,Z 425.704,A -85,B 0,C 180,E1 -16505.023,E2 -16505.023} C_VEL
LIN {X 0,Y 314.526,Z 395.895,A -85,B 0,C 180,E1 -16505.728,E2 -16505.728} C_VEL
LIN {X 0,Y 315.937,Z 352.247,A -85,B 0,C 180,E1 -16506.711,E2 -16506.711} C_VEL
LIN {X 0,Y 308.577,Z 335.385,A -85,B 0,C 180,E1 -16507.979,E2 -16507.979} C_VEL
LIN {X 0,Y 300.986,Z 320.594,A -85,B 0,C 180,E1 -16509.302,E2 -16509.302} C_VEL
LIN {X 0,Y 299.505,Z 317.526,A -85,B 0,C 180,E1 -16509.603,E2 -16509.603} C_VEL
LIN {X 0,Y 298.386,Z 313.318,A -85,B 0,C 180,E1 -16511.262,E2 -16511.262} C_VEL
LIN {X 0,Y 298.354,Z 313.32,A -85,B 0,C 180,E1 -16515.035,E2 -16515.035} C_VEL
LIN {X 0,Y 298.356,Z 313.317,A -85,B 0,C 180,E1 -16516.41,E2 -16516.41} C_VEL
LIN {X 0,Y 297.735,Z 313.399,A -85,B 0,C 180,E1 -16517.537,E2 -16517.537} C_VEL
LIN {X 0,Y 294.867,Z 313.754,A -85,B 0,C 180,E1 -16519.372,E2 -16519.372} C_VEL
LIN {X 0,Y 292.426,Z 314.058,A -85,B 0,C 180,E1 -16520.862,E2 -16520.862} C_VEL
LIN {X 0,Y 291.411,Z 314.18,A -85,B 0,C 180,E1 -16522.017,E2 -16522.017} C_VEL
LIN {X 0,Y 291.348,Z 314.188,A -85,B 0,C 180,E1 -16522.408,E2 -16522.408} C_VEL
LIN {X 0,Y 291.345,Z 314.187,A -85,B 0,C 180,E1 -16526.302,E2 -16526.302} C_VEL
LIN {X 0,Y 291.387,Z 314.179,A -85,B 0,C 180,E1 -16530.26,E2 -16530.26} C_VEL
LIN {X 0,Y 291.416,Z 314.178,A -85,B 0,C 180,E1 -16534.272,E2 -16534.272} C_VEL
LIN {X 0,Y 291.374,Z 314.18,A -85,B 0,C 180,E1 -16537.299,E2 -16537.299} C_VEL
LIN {X 0,Y 291.458,Z 314.168,A -85,B 0,C 180,E1 -16540.27,E2 -16540.27} C_VEL
LIN {X 0,Y 291.556,Z 314.158,A -85,B 0,C 180,E1 -16544.624,E2 -16544.624} C_VEL
LIN {X 0,Y 291.537,Z 314.161,A -85,B 0,C 180,E1 -16548.881,E2 -16548.881} C_VEL
LIN {X 0,Y 291.71,Z 314.149,A -85,B 0,C 180,E1 -16551.689,E2 -16551.689} C_VEL
LIN {X 0,Y 291.63,Z 314.154,A -85,B 0,C 180,E1 -16554.469,E2 -16554.469} C_VEL
LIN {X 0,Y 291.889,Z 314.118,A -85,B 0,C 180,E1 -16558.621,E2 -16558.621} C_VEL
LIN {X 0,Y 291.888,Z 314.122,A -85,B 0,C 180,E1 -16561.38,E2 -16561.38} C_VEL
LIN {X 0,Y 291.746,Z 314.13,A -85,B 0,C 180,E1 -16566.918,E2 -16566.918} C_VEL
LIN {X 0,Y 291.63,Z 314.155,A -85,B 0,C 180,E1 -16569.712,E2 -16569.712} C_VEL
LIN {X 0,Y 291.523,Z 314.169,A -85,B 0,C 180,E1 -16573.951,E2 -16573.951} C_VEL
LIN {X 0,Y 291.488,Z 314.168,A -85,B 0,C 180,E1 -16576.818,E2 -16576.818} C_VEL
LIN {X 0,Y 291.452,Z 314.173,A -85,B 0,C 180,E1 -16579.875,E2 -16579.875} C_VEL
LIN {X 0,Y 291.384,Z 314.182,A -85,B 0,C 180,E1 -16584.207,E2 -16584.207} C_VEL
LIN {X 0,Y 291.427,Z 314.181,A -85,B 0,C 180,E1 -16587.271,E2 -16587.271} C_VEL
LIN {X 0,Y 291.339,Z 314.194,A -85,B 0,C 180,E1 -16590.437,E2 -16590.437} C_VEL
LIN {X 0,Y 291.346,Z 314.193,A -85,B 0,C 180,E1 -16593.699,E2 -16593.699} C_VEL
LIN {X 0,Y 291.378,Z 314.189,A -85,B 0,C 180,E1 -16597.254,E2 -16597.254} C_VEL
LIN {X 0,Y 291.334,Z 314.169,A -85,B 0,C 180,E1 -16600.643,E2 -16600.643} C_VEL
LIN {X 0,Y 291.292,Z 314.196,A -85,B 0,C 180,E1 -16604.402,E2 -16604.402} C_VEL
LIN {X 0,Y 291.328,Z 314.195,A -85,B 0,C 180,E1 -16608.404,E2 -16608.404} C_VEL
LIN {X 0,Y 291.382,Z 314.183,A -85,B 0,C 180,E1 -16612.311,E2 -16612.311} C_VEL
LIN {X 0,Y 294.13,Z 324.783,A -85,B 0,C 180,E1 -16616.253,E2 -16616.253} C_VEL
LIN {X 0,Y 296.549,Z 335.112,A -85,B 0,C 180,E1 -16619.803,E2 -16619.803} C_VEL
LIN {X 0,Y 296.815,Z 336.349,A -85,B 0,C 180,E1 -16620.152,E2 -16620.152} C_VEL
LIN {X 0,Y 302.529,Z 349.156,A -85,B 0,C 180,E1 -16621.219,E2 -16621.219} C_VEL
LIN {X 0,Y 307.287,Z 372.965,A -85,B 0,C 180,E1 -16622.421,E2 -16622.421} C_VEL
LIN {X 0,Y 308.941,Z 384.275,A -85,B 0,C 180,E1 -16622.907,E2 -16622.907} C_VEL
LIN {X 0,Y 306.965,Z 445.331,A -85,B 0,C 180,E1 -16624.351,E2 -16624.351} C_VEL
LIN {X 0,Y 305.929,Z 458.42,A -85,B 0,C 180,E1 -16624.895,E2 -16624.895} C_VEL
LIN {X 0,Y 304.516,Z 470.488,A -85,B 0,C 180,E1 -16625.635,E2 -16625.635} C_VEL
LIN {X 0,Y 302.875,Z 481.882,A -85,B 0,C 180,E1 -16626.586,E2 -16626.586} C_VEL
LIN {X 0,Y 300.832,Z 493.602,A -85,B 0,C 180,E1 -16627.87,E2 -16627.87} C_VEL
LIN {X 0,Y 298.714,Z 504.125,A -85,B 0,C 180,E1 -16629.334,E2 -16629.334} C_VEL
LIN {X 0,Y 296.624,Z 513.631,A -85,B 0,C 180,E1 -16630.987,E2 -16630.987} C_VEL
LIN {X 0,Y 294.69,Z 522.444,A -85,B 0,C 180,E1 -16632.919,E2 -16632.919} C_VEL
LIN {X 0,Y 293.006,Z 530.201,A -85,B 0,C 180,E1 -16635.057,E2 -16635.057} C_VEL
LIN {X 0,Y 291.342,Z 537.053,A -85,B 0,C 180,E1 -16637.461,E2 -16637.461} C_VEL
LIN {X 0,Y 290.468,Z 541.596,A -85,B 0,C 180,E1 -16639.544,E2 -16639.544} C_VEL
LIN {X 0,Y 289.881,Z 545.071,A -85,B 0,C 180,E1 -16641.635,E2 -16641.635} C_VEL
LIN {X 0,Y 289.481,Z 548.158,A -85,B 0,C 180,E1 -16644.427,E2 -16644.427} C_VEL
LIN {X 0,Y 289.474,Z 549.674,A -85,B 0,C 180,E1 -16647.216,E2 -16647.216} C_VEL
LIN {X 0,Y 289.445,Z 549.8,A -85,B 0,C 180,E1 -16648.608,E2 -16648.608} C_VEL
LIN {X 0,Y 289.495,Z 549.537,A -85,B 0,C 180,E1 -16650,E2 -16650} C_VEL
LIN {X 0,Y 289.469,Z 548.881,A -85,B 0,C 180,E1 -16651.391,E2 -16651.391} C_VEL
LIN {X 0,Y 289.497,Z 547.831,A -85,B 0,C 180,E1 -16652.782,E2 -16652.782} C_VEL
LIN {X 0,Y 289.486,Z 546.319,A -85,B 0,C 180,E1 -16654.176,E2 -16654.176} C_VEL
LIN {X 0,Y 289.569,Z 543.25,A -85,B 0,C 180,E1 -16656.27,E2 -16656.27} C_VEL
LIN {X 0,Y 289.828,Z 539.105,A -85,B 0,C 180,E1 -16658.365,E2 -16658.365} C_VEL
LIN {X 0,Y 290.386,Z 532.745,A -85,B 0,C 180,E1 -16660.81,E2 -16660.81} C_VEL
LIN {X 0,Y 291.222,Z 525.812,A -85,B 0,C 180,E1 -16662.898,E2 -16662.898} C_VEL
LIN {X 0,Y 292.132,Z 518.722,A -85,B 0,C 180,E1 -16664.631,E2 -16664.631} C_VEL
LIN {X 0,Y 293.368,Z 509.708,A -85,B 0,C 180,E1 -16666.433,E2 -16666.433} C_VEL
LIN {X 0,Y 294.565,Z 499.558,A -85,B 0,C 180,E1 -16668.069,E2 -16668.069} C_VEL
LIN {X 0,Y 295.917,Z 489.065,A -85,B 0,C 180,E1 -16669.42,E2 -16669.42} C_VEL
LIN {X 0,Y 297.242,Z 477.529,A -85,B 0,C 180,E1 -16670.591,E2 -16670.591} C_VEL
LIN {X 0,Y 298.392,Z 465.573,A -85,B 0,C 180,E1 -16671.502,E2 -16671.502} C_VEL
LIN {X 0,Y 299.358,Z 452.663,A -85,B 0,C 180,E1 -16672.199,E2 -16672.199} C_VEL
LIN {X 0,Y 299.847,Z 440.647,A -85,B 0,C 180,E1 -16672.614,E2 -16672.614} C_VEL
LIN {X 0,Y 301.12,Z 381.057,A -85,B 0,C 180,E1 -16674.02,E2 -16674.02} C_VEL
LIN {X 0,Y 296.008,Z 342.359,A -85,B 0,C 180,E1 -16675.37,E2 -16675.37} C_VEL
LIN {X 0,Y 295.202,Z 336.961,A -85,B 0,C 180,E1 -16675.581,E2 -16675.581} C_VEL
LIN {X 0,Y 295.346,Z 333.671,A -85,B 0,C 180,E1 -16676.497,E2 -16676.497} C_VEL
LIN {X 0,Y 293.104,Z 321.995,A -85,B 0,C 180,E1 -16680.019,E2 -16680.019} C_VEL
LIN {X 0,Y 291.362,Z 314.194,A -85,B 0,C 180,E1 -16682.537,E2 -16682.537} C_VEL
LIN {X 0,Y 291.361,Z 314.191,A -85,B 0,C 180,E1 -16685.373,E2 -16685.373} C_VEL
LIN {X 0,Y 291.363,Z 314.191,A -85,B 0,C 180,E1 -16688.839,E2 -16688.839} C_VEL
LIN {X 0,Y 291.319,Z 314.199,A -85,B 0,C 180,E1 -16692.491,E2 -16692.491} C_VEL
LIN {X 0,Y 291.308,Z 314.2,A -85,B 0,C 180,E1 -16696.365,E2 -16696.365} C_VEL
LIN {X 0,Y 291.376,Z 314.192,A -85,B 0,C 180,E1 -16700.518,E2 -16700.518} C_VEL
LIN {X 0,Y 291.402,Z 314.189,A -85,B 0,C 180,E1 -16702.918,E2 -16702.918} C_VEL
LIN {X 0,Y 291.342,Z 314.194,A -85,B 0,C 180,E1 -16706.301,E2 -16706.301} C_VEL
LIN {X 0,Y 291.381,Z 314.188,A -85,B 0,C 180,E1 -16710.261,E2 -16710.261} C_VEL
LIN {X 0,Y 291.409,Z 314.184,A -85,B 0,C 180,E1 -16714.271,E2 -16714.271} C_VEL
LIN {X 0,Y 291.378,Z 314.19,A -85,B 0,C 180,E1 -16717.299,E2 -16717.299} C_VEL
LIN {X 0,Y 291.455,Z 314.177,A -85,B 0,C 180,E1 -16720.27,E2 -16720.27} C_VEL
LIN {X 0,Y 291.552,Z 314.166,A -85,B 0,C 180,E1 -16724.623,E2 -16724.623} C_VEL
LIN {X 0,Y 291.533,Z 314.161,A -85,B 0,C 180,E1 -16728.88,E2 -16728.88} C_VEL
LIN {X 0,Y 291.703,Z 314.149,A -85,B 0,C 180,E1 -16731.688,E2 -16731.688} C_VEL
LIN {X 0,Y 291.624,Z 314.156,A -85,B 0,C 180,E1 -16734.468,E2 -16734.468} C_VEL
LIN {X 0,Y 291.885,Z 314.116,A -85,B 0,C 180,E1 -16738.62,E2 -16738.62} C_VEL
LIN {X 0,Y 291.884,Z 314.121,A -85,B 0,C 180,E1 -16741.379,E2 -16741.379} C_VEL
LIN {X 0,Y 291.654,Z 314.15,A -85,B 0,C 180,E1 -16746.537,E2 -16746.537} C_VEL
LIN {X 0,Y 291.567,Z 314.159,A -85,B 0,C 180,E1 -16749.714,E2 -16749.714} C_VEL
LIN {X 0,Y 291.517,Z 314.172,A -85,B 0,C 180,E1 -16753.95,E2 -16753.95} C_VEL
LIN {X 0,Y 291.481,Z 314.173,A -85,B 0,C 180,E1 -16756.818,E2 -16756.818} C_VEL
LIN {X 0,Y 291.446,Z 314.174,A -85,B 0,C 180,E1 -16759.875,E2 -16759.875} C_VEL
LIN {X 0,Y 291.379,Z 314.189,A -85,B 0,C 180,E1 -16764.207,E2 -16764.207} C_VEL
LIN {X 0,Y 291.418,Z 314.18,A -85,B 0,C 180,E1 -16767.272,E2 -16767.272} C_VEL
LIN {X 0,Y 291.333,Z 314.189,A -85,B 0,C 180,E1 -16770.437,E2 -16770.437} C_VEL
LIN {X 0,Y 291.34,Z 314.191,A -85,B 0,C 180,E1 -16773.699,E2 -16773.699} C_VEL
LIN {X 0,Y 291.367,Z 314.185,A -85,B 0,C 180,E1 -16777.253,E2 -16777.253} C_VEL
LIN {X 0,Y 291.328,Z 314.192,A -85,B 0,C 180,E1 -16780.643,E2 -16780.643} C_VEL
LIN {X 0,Y 291.286,Z 314.198,A -85,B 0,C 180,E1 -16784.402,E2 -16784.402} C_VEL
LIN {X 0,Y 291.291,Z 314.198,A -85,B 0,C 180,E1 -16788.412,E2 -16788.412} C_VEL
LIN {X 0,Y 291.331,Z 314.194,A -85,B 0,C 180,E1 -16791.156,E2 -16791.156} C_VEL
LIN {X 0,Y 291.357,Z 314.191,A -85,B 0,C 180,E1 -16794.626,E2 -16794.626} C_VEL
LIN {X 0,Y 291.363,Z 314.189,A -85,B 0,C 180,E1 -16797.951,E2 -16797.951} C_VEL
LIN {X 0,Y 291.319,Z 314.195,A -85,B 0,C 180,E1 -16801.152,E2 -16801.152} C_VEL
LIN {X 0,Y 291.344,Z 314.191,A -85,B 0,C 180,E1 -16804.266,E2 -16804.266} C_VEL
LIN {X 0,Y 291.359,Z 314.193,A -85,B 0,C 180,E1 -16807.298,E2 -16807.298} C_VEL
LIN {X 0,Y 291.438,Z 314.182,A -85,B 0,C 180,E1 -16810.269,E2 -16810.269} C_VEL
LIN {X 0,Y 291.497,Z 314.186,A -85,B 0,C 180,E1 -16813.265,E2 -16813.265} C_VEL
LIN {X 0,Y 292.143,Z 317.177,A -85,B 0,C 180,E1 -16814.258,E2 -16814.258} C_VEL
LIN {X 0,Y 299.184,Z 336.509,A -85,B 0,C 180,E1 -16815.309,E2 -16815.309} C_VEL
LIN {X 0,Y 300.948,Z 342.943,A -85,B 0,C 180,E1 -16815.602,E2 -16815.602} C_VEL
LIN {X 0,Y 301.837,Z 348.331,A -85,B 0,C 180,E1 -16815.801,E2 -16815.801} C_VEL
LIN {X 0,Y 299.989,Z 424.69,A -85,B 0,C 180,E1 -16817.618,E2 -16817.618} C_VEL
LIN {X 0,Y 299.338,Z 438.459,A -85,B 0,C 180,E1 -16818.231,E2 -16818.231} C_VEL
LIN {X 0,Y 298.527,Z 450.878,A -85,B 0,C 180,E1 -16819.059,E2 -16819.059} C_VEL
LIN {X 0,Y 297.472,Z 462.761,A -85,B 0,C 180,E1 -16820.138,E2 -16820.138} C_VEL
LIN {X 0,Y 296.016,Z 472.936,A -85,B 0,C 180,E1 -16821.295,E2 -16821.295} C_VEL
LIN {X 0,Y 294.819,Z 483.403,A -85,B 0,C 180,E1 -16822.811,E2 -16822.811} C_VEL
LIN {X 0,Y 293.5,Z 492.873,A -85,B 0,C 180,E1 -16824.504,E2 -16824.504} C_VEL
LIN {X 0,Y 292.31,Z 501.966,A -85,B 0,C 180,E1 -16826.555,E2 -16826.555} C_VEL
LIN {X 0,Y 291.23,Z 509.31,A -85,B 0,C 180,E1 -16828.618,E2 -16828.618} C_VEL
LIN {X 0,Y 290.568,Z 515.189,A -85,B 0,C 180,E1 -16830.693,E2 -16830.693} C_VEL
LIN {X 0,Y 289.979,Z 519.846,A -85,B 0,C 180,E1 -16832.779,E2 -16832.779} C_VEL
LIN {X 0,Y 289.807,Z 523.389,A -85,B 0,C 180,E1 -16834.869,E2 -16834.869} C_VEL
LIN {X 0,Y 289.572,Z 525.943,A -85,B 0,C 180,E1 -16836.971,E2 -16836.971} C_VEL
LIN {X 0,Y 289.415,Z 527.146,A -85,B 0,C 180,E1 -16838.378,E2 -16838.378} C_VEL
LIN {X 0,Y 289.371,Z 528.263,A -85,B 0,C 180,E1 -16841.204,E2 -16841.204} C_VEL
LIN {X 0,Y 289.508,Z 528.237,A -85,B 0,C 180,E1 -16842.62,E2 -16842.62} C_VEL
LIN {X 0,Y 289.73,Z 527.805,A -85,B 0,C 180,E1 -16844.039,E2 -16844.039} C_VEL
LIN {X 0,Y 289.937,Z 526.93,A -85,B 0,C 180,E1 -16845.465,E2 -16845.465} C_VEL
LIN {X 0,Y 290.241,Z 525.65,A -85,B 0,C 180,E1 -16846.893,E2 -16846.893} C_VEL
LIN {X 0,Y 290.966,Z 522.904,A -85,B 0,C 180,E1 -16849.031,E2 -16849.031} C_VEL
LIN {X 0,Y 291.94,Z 519.092,A -85,B 0,C 180,E1 -16851.168,E2 -16851.168} C_VEL
LIN {X 0,Y 293.202,Z 514.098,A -85,B 0,C 180,E1 -16853.298,E2 -16853.298} C_VEL
LIN {X 0,Y 294.703,Z 507.761,A -85,B 0,C 180,E1 -16855.421,E2 -16855.421} C_VEL
LIN {X 0,Y 296.651,Z 499.756,A -85,B 0,C 180,E1 -16857.515,E2 -16857.515} C_VEL
LIN {X 0,Y 298.828,Z 490.068,A -85,B 0,C 180,E1 -16859.52,E2 -16859.52} C_VEL
LIN {X 0,Y 300.891,Z 480.3,A -85,B 0,C 180,E1 -16861.117,E2 -16861.117} C_VEL
LIN {X 0,Y 302.679,Z 469.956,A -85,B 0,C 180,E1 -16862.476,E2 -16862.476} C_VEL
LIN {X 0,Y 304.405,Z 458.613,A -85,B 0,C 180,E1 -16863.649,E2 -16863.649} C_VEL
LIN {X 0,Y 305.71,Z 447.058,A -85,B 0,C 180,E1 -16864.579,E2 -16864.579} C_VEL
LIN {X 0,Y 306.698,Z 434.734,A -85,B 0,C 180,E1 -16865.302,E2 -16865.302} C_VEL
LIN {X 0,Y 307.367,Z 424.091,A -85,B 0,C 180,E1 -16865.717,E2 -16865.717} C_VEL
LIN {X 0,Y 309.72,Z 354.031,A -85,B 0,C 180,E1 -16867.347,E2 -16867.347} C_VEL
LIN {X 0,Y 302.717,Z 338.102,A -85,B 0,C 180,E1 -16868.6,E2 -16868.6} C_VEL
LIN {X 0,Y 295.808,Z 324.555,A -85,B 0,C 180,E1 -16869.851,E2 -16869.851} C_VEL
LIN {X 0,Y 292.309,Z 317.86,A -85,B 0,C 180,E1 -16870.535,E2 -16870.535} C_VEL
LIN {X 0,Y 291.312,Z 314.195,A -85,B 0,C 180,E1 -16871.988,E2 -16871.988} C_VEL
LIN {X 0,Y 291.309,Z 314.199,A -85,B 0,C 180,E1 -16876.367,E2 -16876.367} C_VEL
LIN {X 0,Y 291.378,Z 314.187,A -85,B 0,C 180,E1 -16880.519,E2 -16880.519} C_VEL
LIN {X 0,Y 291.348,Z 314.188,A -85,B 0,C 180,E1 -16882.408,E2 -16882.408} C_VEL
LIN {X 0,Y 290.719,Z 314.27,A -85,B 0,C 180,E1 -16883.561,E2 -16883.561} C_VEL
LIN {X 0,Y 287.837,Z 314.626,A -85,B 0,C 180,E1 -16885.437,E2 -16885.437} C_VEL
LIN {X 0,Y 285.382,Z 314.93,A -85,B 0,C 180,E1 -16886.96,E2 -16886.96} C_VEL
LIN {X 0,Y 284.354,Z 315.056,A -85,B 0,C 180,E1 -16888.142,E2 -16888.142} C_VEL
LIN {X 0,Y 284.286,Z 315.06,A -85,B 0,C 180,E1 -16888.542,E2 -16888.542} C_VEL
LIN {X 0,Y 284.332,Z 315.055,A -85,B 0,C 180,E1 -16891.99,E2 -16891.99} C_VEL
LIN {X 0,Y 284.338,Z 315.06,A -85,B 0,C 180,E1 -16895.154,E2 -16895.154} C_VEL
LIN {X 0,Y 284.388,Z 315.05,A -85,B 0,C 180,E1 -16899.898,E2 -16899.898} C_VEL
LIN {X 0,Y 284.492,Z 315.038,A -85,B 0,C 180,E1 -16904.46,E2 -16904.46} C_VEL
LIN {X 0,Y 284.489,Z 315.04,A -85,B 0,C 180,E1 -16908.602,E2 -16908.602} C_VEL
LIN {X 0,Y 284.66,Z 315.027,A -85,B 0,C 180,E1 -16911.481,E2 -16911.481} C_VEL
LIN {X 0,Y 284.601,Z 315.028,A -85,B 0,C 180,E1 -16914.332,E2 -16914.332} C_VEL
LIN {X 0,Y 284.855,Z 314.993,A -85,B 0,C 180,E1 -16918.587,E2 -16918.587} C_VEL
LIN {X 0,Y 284.855,Z 314.998,A -85,B 0,C 180,E1 -16921.414,E2 -16921.414} C_VEL
LIN {X 0,Y 284.698,Z 315.007,A -85,B 0,C 180,E1 -16927.09,E2 -16927.09} C_VEL
LIN {X 0,Y 284.567,Z 315.036,A -85,B 0,C 180,E1 -16929.956,E2 -16929.956} C_VEL
LIN {X 0,Y 284.483,Z 315.048,A -85,B 0,C 180,E1 -16934.303,E2 -16934.303} C_VEL
LIN {X 0,Y 284.427,Z 315.051,A -85,B 0,C 180,E1 -16937.249,E2 -16937.249} C_VEL
LIN {X 0,Y 284.379,Z 315.052,A -85,B 0,C 180,E1 -16940.243,E2 -16940.243} C_VEL
LIN {X 0,Y 284.341,Z 315.058,A -85,B 0,C 180,E1 -16944.847,E2 -16944.847} C_VEL
LIN {X 0,Y 284.336,Z 315.062,A -85,B 0,C 180,E1 -16948.011,E2 -16948.011} C_VEL
LIN {X 0,Y 284.297,Z 315.069,A -85,B 0,C 180,E1 -16951.275,E2 -16951.275} C_VEL
LIN {X 0,Y 284.342,Z 315.059,A -85,B 0,C 180,E1 -16955.348,E2 -16955.348} C_VEL
LIN {X 0,Y 284.314,Z 315.067,A -85,B 0,C 180,E1 -16958.169,E2 -16958.169} C_VEL
LIN {X 0,Y 284.271,Z 315.063,A -85,B 0,C 180,E1 -16962.124,E2 -16962.124} C_VEL
LIN {X 0,Y 284.257,Z 315.076,A -85,B 0,C 180,E1 -16966.189,E2 -16966.189} C_VEL
LIN {X 0,Y 284.309,Z 315.071,A -85,B 0,C 180,E1 -16970.024,E2 -16970.024} C_VEL
LIN {X 0,Y 284.326,Z 315.082,A -85,B 0,C 180,E1 -16971.494,E2 -16971.494} C_VEL
LIN {X 0,Y 286.951,Z 324.966,A -85,B 0,C 180,E1 -16975.312,E2 -16975.312} C_VEL
LIN {X 0,Y 289.428,Z 335.468,A -85,B 0,C 180,E1 -16979.06,E2 -16979.06} C_VEL
LIN {X 0,Y 289.67,Z 336.314,A -85,B 0,C 180,E1 -16979.21,E2 -16979.21} C_VEL
LIN {X 0,Y 296.889,Z 352.181,A -85,B 0,C 180,E1 -16980.612,E2 -16980.612} C_VEL
LIN {X 0,Y 301.54,Z 376.058,A -85,B 0,C 180,E1 -16981.845,E2 -16981.845} C_VEL
LIN {X 0,Y 302.841,Z 384.967,A -85,B 0,C 180,E1 -16982.241,E2 -16982.241} C_VEL
LIN {X 0,Y 300.801,Z 445.189,A -85,B 0,C 180,E1 -16983.692,E2 -16983.692} C_VEL
LIN {X 0,Y 299.641,Z 458.995,A -85,B 0,C 180,E1 -16984.284,E2 -16984.284} C_VEL
LIN {X 0,Y 298.109,Z 471.397,A -85,B 0,C 180,E1 -16985.076,E2 -16985.076} C_VEL
LIN {X 0,Y 296.402,Z 482.476,A -85,B 0,C 180,E1 -16986.043,E2 -16986.043} C_VEL
LIN {X 0,Y 294.281,Z 494.016,A -85,B 0,C 180,E1 -16987.35,E2 -16987.35} C_VEL
LIN {X 0,Y 292.105,Z 504.422,A -85,B 0,C 180,E1 -16988.844,E2 -16988.844} C_VEL
LIN {X 0,Y 289.939,Z 513.818,A -85,B 0,C 180,E1 -16990.531,E2 -16990.531} C_VEL
LIN {X 0,Y 287.845,Z 522.779,A -85,B 0,C 180,E1 -16992.566,E2 -16992.566} C_VEL
LIN {X 0,Y 286.15,Z 530.23,A -85,B 0,C 180,E1 -16994.691,E2 -16994.691} C_VEL
LIN {X 0,Y 284.382,Z 537,A -85,B 0,C 180,E1 -16997.148,E2 -16997.148} C_VEL
LIN {X 0,Y 283.478,Z 541.493,A -85,B 0,C 180,E1 -16999.284,E2 -16999.284} C_VEL
LIN {X 0,Y 282.827,Z 544.926,A -85,B 0,C 180,E1 -17001.425,E2 -17001.425} C_VEL
LIN {X 0,Y 282.388,Z 547.964,A -85,B 0,C 180,E1 -17004.286,E2 -17004.286} C_VEL
LIN {X 0,Y 282.339,Z 548.897,A -85,B 0,C 180,E1 -17005.717,E2 -17005.717} C_VEL
LIN {X 0,Y 282.378,Z 549.425,A -85,B 0,C 180,E1 -17007.146,E2 -17007.146} C_VEL
LIN {X 0,Y 282.367,Z 549.526,A -85,B 0,C 180,E1 -17008.573,E2 -17008.573} C_VEL
LIN {X 0,Y 282.412,Z 549.242,A -85,B 0,C 180,E1 -17009.999,E2 -17009.999} C_VEL
LIN {X 0,Y 282.391,Z 548.567,A -85,B 0,C 180,E1 -17011.426,E2 -17011.426} C_VEL
LIN {X 0,Y 282.424,Z 547.485,A -85,B 0,C 180,E1 -17012.852,E2 -17012.852} C_VEL
LIN {X 0,Y 282.436,Z 544.249,A -85,B 0,C 180,E1 -17015.529,E2 -17015.529} C_VEL
LIN {X 0,Y 282.666,Z 540.151,A -85,B 0,C 180,E1 -17017.859,E2 -17017.859} C_VEL
LIN {X 0,Y 283.075,Z 535.181,A -85,B 0,C 180,E1 -17020.008,E2 -17020.008} C_VEL
LIN {X 0,Y 283.74,Z 528.911,A -85,B 0,C 180,E1 -17022.153,E2 -17022.153} C_VEL
LIN {X 0,Y 284.841,Z 521.082,A -85,B 0,C 180,E1 -17024.284,E2 -17024.284} C_VEL
LIN {X 0,Y 286.143,Z 511.948,A -85,B 0,C 180,E1 -17026.266,E2 -17026.266} C_VEL
LIN {X 0,Y 287.326,Z 502.16,A -85,B 0,C 180,E1 -17027.987,E2 -17027.987} C_VEL
LIN {X 0,Y 288.769,Z 490.92,A -85,B 0,C 180,E1 -17029.55,E2 -17029.55} C_VEL
LIN {X 0,Y 290.162,Z 479.905,A -85,B 0,C 180,E1 -17030.746,E2 -17030.746} C_VEL
LIN {X 0,Y 291.418,Z 467.703,A -85,B 0,C 180,E1 -17031.764,E2 -17031.764} C_VEL
LIN {X 0,Y 292.44,Z 455.045,A -85,B 0,C 180,E1 -17032.52,E2 -17032.52} C_VEL
LIN {X 0,Y 293.132,Z 442.027,A -85,B 0,C 180,E1 -17033.013,E2 -17033.013} C_VEL
LIN {X 0,Y 294.43,Z 381.267,A -85,B 0,C 180,E1 -17034.489,E2 -17034.489} C_VEL
LIN {X 0,Y 289.274,Z 342.317,A -85,B 0,C 180,E1 -17035.893,E2 -17035.893} C_VEL
LIN {X 0,Y 288.408,Z 336.56,A -85,B 0,C 180,E1 -17036.161,E2 -17036.161} C_VEL
LIN {X 0,Y 287.796,Z 331.604,A -85,B 0,C 180,E1 -17037.643,E2 -17037.643} C_VEL
LIN {X 0,Y 285.501,Z 320.51,A -85,B 0,C 180,E1 -17041.127,E2 -17041.127} C_VEL
LIN {X 0,Y 284.324,Z 315.07,A -85,B 0,C 180,E1 -17042.942,E2 -17042.942} C_VEL
LIN {X 0,Y 284.334,Z 315.069,A -85,B 0,C 180,E1 -17046.385,E2 -17046.385} C_VEL
LIN {X 0,Y 284.305,Z 315.071,A -85,B 0,C 180,E1 -17049.994,E2 -17049.994} C_VEL
LIN {X 0,Y 284.244,Z 315.079,A -85,B 0,C 180,E1 -17054.19,E2 -17054.19} C_VEL
LIN {X 0,Y 284.27,Z 315.075,A -85,B 0,C 180,E1 -17058.124,E2 -17058.124} C_VEL
LIN {X 0,Y 284.317,Z 315.07,A -85,B 0,C 180,E1 -17062.278,E2 -17062.278} C_VEL
LIN {X 0,Y 284.306,Z 315.07,A -85,B 0,C 180,E1 -17065.35,E2 -17065.35} C_VEL
LIN {X 0,Y 284.291,Z 315.074,A -85,B 0,C 180,E1 -17068.725,E2 -17068.725} C_VEL
LIN {X 0,Y 284.391,Z 315.062,A -85,B 0,C 180,E1 -17072.827,E2 -17072.827} C_VEL
LIN {X 0,Y 284.363,Z 315.063,A -85,B 0,C 180,E1 -17076.706,E2 -17076.706} C_VEL
LIN {X 0,Y 284.401,Z 315.06,A -85,B 0,C 180,E1 -17081.261,E2 -17081.261} C_VEL
LIN {X 0,Y 284.489,Z 315.045,A -85,B 0,C 180,E1 -17084.459,E2 -17084.459} C_VEL
LIN {X 0,Y 284.484,Z 315.037,A -85,B 0,C 180,E1 -17088.601,E2 -17088.601} C_VEL
LIN {X 0,Y 284.653,Z 315.025,A -85,B 0,C 180,E1 -17091.481,E2 -17091.481} C_VEL
LIN {X 0,Y 284.594,Z 315.032,A -85,B 0,C 180,E1 -17094.331,E2 -17094.331} C_VEL
LIN {X 0,Y 284.851,Z 314.991,A -85,B 0,C 180,E1 -17098.586,E2 -17098.586} C_VEL
LIN {X 0,Y 284.85,Z 314.997,A -85,B 0,C 180,E1 -17101.413,E2 -17101.413} C_VEL
LIN {X 0,Y 284.649,Z 315.023,A -85,B 0,C 180,E1 -17107.091,E2 -17107.091} C_VEL
LIN {X 0,Y 284.513,Z 315.036,A -85,B 0,C 180,E1 -17109.957,E2 -17109.957} C_VEL
LIN {X 0,Y 284.477,Z 315.05,A -85,B 0,C 180,E1 -17114.303,E2 -17114.303} C_VEL
LIN {X 0,Y 284.418,Z 315.052,A -85,B 0,C 180,E1 -17117.248,E2 -17117.248} C_VEL
LIN {X 0,Y 284.373,Z 315.054,A -85,B 0,C 180,E1 -17120.242,E2 -17120.242} C_VEL
LIN {X 0,Y 284.334,Z 315.066,A -85,B 0,C 180,E1 -17124.847,E2 -17124.847} C_VEL
LIN {X 0,Y 284.328,Z 315.065,A -85,B 0,C 180,E1 -17128.011,E2 -17128.011} C_VEL
LIN {X 0,Y 284.291,Z 315.065,A -85,B 0,C 180,E1 -17131.275,E2 -17131.275} C_VEL
LIN {X 0,Y 284.336,Z 315.064,A -85,B 0,C 180,E1 -17135.348,E2 -17135.348} C_VEL
LIN {X 0,Y 284.304,Z 315.064,A -85,B 0,C 180,E1 -17138.17,E2 -17138.17} C_VEL
LIN {X 0,Y 284.265,Z 315.072,A -85,B 0,C 180,E1 -17142.125,E2 -17142.125} C_VEL
LIN {X 0,Y 284.233,Z 315.071,A -85,B 0,C 180,E1 -17146.186,E2 -17146.186} C_VEL
LIN {X 0,Y 284.279,Z 315.071,A -85,B 0,C 180,E1 -17150.03,E2 -17150.03} C_VEL
LIN {X 0,Y 284.325,Z 315.068,A -85,B 0,C 180,E1 -17153.614,E2 -17153.614} C_VEL
LIN {X 0,Y 284.303,Z 315.072,A -85,B 0,C 180,E1 -17157.191,E2 -17157.191} C_VEL
LIN {X 0,Y 284.31,Z 315.065,A -85,B 0,C 180,E1 -17160.371,E2 -17160.371} C_VEL
LIN {X 0,Y 284.295,Z 315.072,A -85,B 0,C 180,E1 -17163.579,E2 -17163.579} C_VEL
LIN {X 0,Y 284.318,Z 315.067,A -85,B 0,C 180,E1 -17166.704,E2 -17166.704} C_VEL
LIN {X 0,Y 284.374,Z 315.063,A -85,B 0,C 180,E1 -17169.905,E2 -17169.905} C_VEL
LIN {X 0,Y 284.463,Z 315.248,A -85,B 0,C 180,E1 -17172.921,E2 -17172.921} C_VEL
LIN {X 0,Y 284.952,Z 317.468,A -85,B 0,C 180,E1 -17173.679,E2 -17173.679} C_VEL
LIN {X 0,Y 292.566,Z 338.02,A -85,B 0,C 180,E1 -17174.843,E2 -17174.843} C_VEL
LIN {X 0,Y 294.405,Z 344.305,A -85,B 0,C 180,E1 -17175.148,E2 -17175.148} C_VEL
LIN {X 0,Y 295.158,Z 349.957,A -85,B 0,C 180,E1 -17175.351,E2 -17175.351} C_VEL
LIN {X 0,Y 293.277,Z 425.449,A -85,B 0,C 180,E1 -17177.194,E2 -17177.194} C_VEL
LIN {X 0,Y 292.599,Z 439.126,A -85,B 0,C 180,E1 -17177.824,E2 -17177.824} C_VEL
LIN {X 0,Y 291.72,Z 451.932,A -85,B 0,C 180,E1 -17178.712,E2 -17178.712} C_VEL
LIN {X 0,Y 290.552,Z 464.409,A -85,B 0,C 180,E1 -17179.901,E2 -17179.901} C_VEL
LIN {X 0,Y 289.032,Z 474.337,A -85,B 0,C 180,E1 -17181.083,E2 -17181.083} C_VEL
LIN {X 0,Y 287.816,Z 484.608,A -85,B 0,C 180,E1 -17182.635,E2 -17182.635} C_VEL
LIN {X 0,Y 286.471,Z 493.871,A -85,B 0,C 180,E1 -17184.369,E2 -17184.369} C_VEL
LIN {X 0,Y 285.242,Z 502.831,A -85,B 0,C 180,E1 -17186.469,E2 -17186.469} C_VEL
LIN {X 0,Y 284.135,Z 510.072,A -85,B 0,C 180,E1 -17188.583,E2 -17188.583} C_VEL
LIN {X 0,Y 283.463,Z 515.854,A -85,B 0,C 180,E1 -17190.711,E2 -17190.711} C_VEL
LIN {X 0,Y 282.877,Z 520.423,A -85,B 0,C 180,E1 -17192.849,E2 -17192.849} C_VEL
LIN {X 0,Y 282.786,Z 522.824,A -85,B 0,C 180,E1 -17194.276,E2 -17194.276} C_VEL
LIN {X 0,Y 282.662,Z 525.152,A -85,B 0,C 180,E1 -17195.99,E2 -17195.99} C_VEL
LIN {X 0,Y 282.304,Z 527.508,A -85,B 0,C 180,E1 -17198.591,E2 -17198.591} C_VEL
LIN {X 0,Y 282.318,Z 528.548,A -85,B 0,C 180,E1 -17201.488,E2 -17201.488} C_VEL
LIN {X 0,Y 282.659,Z 528.111,A -85,B 0,C 180,E1 -17204.143,E2 -17204.143} C_VEL
LIN {X 0,Y 282.938,Z 527.071,A -85,B 0,C 180,E1 -17205.857,E2 -17205.857} C_VEL
LIN {X 0,Y 283.268,Z 525.755,A -85,B 0,C 180,E1 -17207.321,E2 -17207.321} C_VEL
LIN {X 0,Y 283.799,Z 524.004,A -85,B 0,C 180,E1 -17208.78,E2 -17208.78} C_VEL
LIN {X 0,Y 284.736,Z 520.479,A -85,B 0,C 180,E1 -17210.971,E2 -17210.971} C_VEL
LIN {X 0,Y 285.985,Z 515.793,A -85,B 0,C 180,E1 -17213.154,E2 -17213.154} C_VEL
LIN {X 0,Y 287.675,Z 509.148,A -85,B 0,C 180,E1 -17215.532,E2 -17215.532} C_VEL
LIN {X 0,Y 289.479,Z 502.269,A -85,B 0,C 180,E1 -17217.47,E2 -17217.47} C_VEL
LIN {X 0,Y 291.586,Z 493.555,A -85,B 0,C 180,E1 -17219.447,E2 -17219.447} C_VEL
LIN {X 0,Y 293.699,Z 484.009,A -85,B 0,C 180,E1 -17221.163,E2 -17221.163} C_VEL
LIN {X 0,Y 295.832,Z 473.176,A -85,B 0,C 180,E1 -17222.716,E2 -17222.716} C_VEL
LIN {X 0,Y 297.563,Z 462.748,A -85,B 0,C 180,E1 -17223.904,E2 -17223.904} C_VEL
LIN {X 0,Y 299.116,Z 451.088,A -85,B 0,C 180,E1 -17224.939,E2 -17224.939} C_VEL
LIN {X 0,Y 300.232,Z 439.438,A -85,B 0,C 180,E1 -17225.715,E2 -17225.715} C_VEL
LIN {X 0,Y 301.028,Z 427.042,A -85,B 0,C 180,E1 -17226.289,E2 -17226.289} C_VEL
LIN {X 0,Y 301.994,Z 405.419,A -85,B 0,C 180,E1 -17226.833,E2 -17226.833} C_VEL
LIN {X 0,Y 303.709,Z 356.218,A -85,B 0,C 180,E1 -17227.981,E2 -17227.981} C_VEL
LIN {X 0,Y 296.757,Z 340.415,A -85,B 0,C 180,E1 -17229.274,E2 -17229.274} C_VEL
LIN {X 0,Y 288.933,Z 325.282,A -85,B 0,C 180,E1 -17230.754,E2 -17230.754} C_VEL
LIN {X 0,Y 285.098,Z 318.188,A -85,B 0,C 180,E1 -17231.535,E2 -17231.535} C_VEL
LIN {X 0,Y 284.267,Z 315.075,A -85,B 0,C 180,E1 -17232.801,E2 -17232.801} C_VEL
LIN {X 0,Y 284.255,Z 315.077,A -85,B 0,C 180,E1 -17236.19,E2 -17236.19} C_VEL
LIN {X 0,Y 284.306,Z 315.068,A -85,B 0,C 180,E1 -17240.024,E2 -17240.024} C_VEL
LIN {X 0,Y 284.33,Z 315.062,A -85,B 0,C 180,E1 -17243.614,E2 -17243.614} C_VEL
LIN {X 0,Y 284.308,Z 315.065,A -85,B 0,C 180,E1 -17247.19,E2 -17247.19} C_VEL
LIN {X 0,Y 284.286,Z 315.06,A -85,B 0,C 180,E1 -17248.542,E2 -17248.542} C_VEL
LIN {X 0,Y 283.67,Z 315.139,A -85,B 0,C 180,E1 -17249.726,E2 -17249.726} C_VEL
LIN {X 0,Y 280.864,Z 315.496,A -85,B 0,C 180,E1 -17251.656,E2 -17251.656} C_VEL
LIN {X 0,Y 278.444,Z 315.798,A -85,B 0,C 180,E1 -17253.223,E2 -17253.223} C_VEL
LIN {X 0,Y 277.385,Z 315.926,A -85,B 0,C 180,E1 -17254.437,E2 -17254.437} C_VEL
LIN {X 0,Y 277.289,Z 315.934,A -85,B 0,C 180,E1 -17254.848,E2 -17254.848} C_VEL
LIN {X 0,Y 277.344,Z 315.929,A -85,B 0,C 180,E1 -17259.651,E2 -17259.651} C_VEL
LIN {X 0,Y 277.444,Z 315.916,A -85,B 0,C 180,E1 -17264.278,E2 -17264.278} C_VEL
LIN {X 0,Y 277.435,Z 315.919,A -85,B 0,C 180,E1 -17268.308,E2 -17268.308} C_VEL
LIN {X 0,Y 277.616,Z 315.903,A -85,B 0,C 180,E1 -17271.264,E2 -17271.264} C_VEL
LIN {X 0,Y 277.572,Z 315.902,A -85,B 0,C 180,E1 -17274.188,E2 -17274.188} C_VEL
LIN {X 0,Y 277.821,Z 315.869,A -85,B 0,C 180,E1 -17278.551,E2 -17278.551} C_VEL
LIN {X 0,Y 277.821,Z 315.873,A -85,B 0,C 180,E1 -17281.45,E2 -17281.45} C_VEL
LIN {X 0,Y 277.653,Z 315.885,A -85,B 0,C 180,E1 -17287.271,E2 -17287.271} C_VEL
LIN {X 0,Y 277.508,Z 315.913,A -85,B 0,C 180,E1 -17290.212,E2 -17290.212} C_VEL
LIN {X 0,Y 277.436,Z 315.921,A -85,B 0,C 180,E1 -17294.674,E2 -17294.674} C_VEL
LIN {X 0,Y 277.346,Z 315.932,A -85,B 0,C 180,E1 -17299.234,E2 -17299.234} C_VEL
LIN {X 0,Y 277.294,Z 315.937,A -85,B 0,C 180,E1 -17304.158,E2 -17304.158} C_VEL
LIN {X 0,Y 277.329,Z 315.936,A -85,B 0,C 180,E1 -17307.506,E2 -17307.506} C_VEL
LIN {X 0,Y 277.274,Z 315.947,A -85,B 0,C 180,E1 -17310.482,E2 -17310.482} C_VEL
LIN {X 0,Y 277.249,Z 315.949,A -85,B 0,C 180,E1 -17313.896,E2 -17313.896} C_VEL
LIN {X 0,Y 277.27,Z 315.947,A -85,B 0,C 180,E1 -17317.469,E2 -17317.469} C_VEL
LIN {X 0,Y 277.211,Z 315.93,A -85,B 0,C 180,E1 -17321.237,E2 -17321.237} C_VEL
LIN {X 0,Y 277.203,Z 315.954,A -85,B 0,C 180,E1 -17325.227,E2 -17325.227} C_VEL
LIN {X 0,Y 277.225,Z 315.954,A -85,B 0,C 180,E1 -17329.512,E2 -17329.512} C_VEL
LIN {X 0,Y 277.307,Z 316.024,A -85,B 0,C 180,E1 -17330.63,E2 -17330.63} C_VEL
LIN {X 0,Y 279.559,Z 324.352,A -85,B 0,C 180,E1 -17333.997,E2 -17333.997} C_VEL
LIN {X 0,Y 282.085,Z 334.776,A -85,B 0,C 180,E1 -17337.898,E2 -17337.898} C_VEL
LIN {X 0,Y 282.308,Z 335.759,A -85,B 0,C 180,E1 -17338.16,E2 -17338.16} C_VEL
LIN {X 0,Y 290.046,Z 352.225,A -85,B 0,C 180,E1 -17339.73,E2 -17339.73} C_VEL
LIN {X 0,Y 291.517,Z 356.202,A -85,B 0,C 180,E1 -17340.04,E2 -17340.04} C_VEL
LIN {X 0,Y 295.666,Z 378.216,A -85,B 0,C 180,E1 -17341.199,E2 -17341.199} C_VEL
LIN {X 0,Y 296.759,Z 386.304,A -85,B 0,C 180,E1 -17341.56,E2 -17341.56} C_VEL
LIN {X 0,Y 294.665,Z 445.208,A -85,B 0,C 180,E1 -17343.009,E2 -17343.009} C_VEL
LIN {X 0,Y 293.473,Z 458.846,A -85,B 0,C 180,E1 -17343.606,E2 -17343.606} C_VEL
LIN {X 0,Y 291.882,Z 471.21,A -85,B 0,C 180,E1 -17344.411,E2 -17344.411} C_VEL
LIN {X 0,Y 289.969,Z 483.051,A -85,B 0,C 180,E1 -17345.477,E2 -17345.477} C_VEL
LIN {X 0,Y 287.762,Z 494.435,A -85,B 0,C 180,E1 -17346.807,E2 -17346.807} C_VEL
LIN {X 0,Y 285.509,Z 504.719,A -85,B 0,C 180,E1 -17348.331,E2 -17348.331} C_VEL
LIN {X 0,Y 283.251,Z 513.985,A -85,B 0,C 180,E1 -17350.052,E2 -17350.052} C_VEL
LIN {X 0,Y 281.015,Z 523.106,A -85,B 0,C 180,E1 -17352.193,E2 -17352.193} C_VEL
LIN {X 0,Y 279.301,Z 530.258,A -85,B 0,C 180,E1 -17354.306,E2 -17354.306} C_VEL
LIN {X 0,Y 277.436,Z 536.947,A -85,B 0,C 180,E1 -17356.821,E2 -17356.821} C_VEL
LIN {X 0,Y 276.475,Z 541.39,A -85,B 0,C 180,E1 -17359.009,E2 -17359.009} C_VEL
LIN {X 0,Y 275.794,Z 544.777,A -85,B 0,C 180,E1 -17361.205,E2 -17361.205} C_VEL
LIN {X 0,Y 275.302,Z 547.772,A -85,B 0,C 180,E1 -17364.139,E2 -17364.139} C_VEL
LIN {X 0,Y 275.25,Z 548.684,A -85,B 0,C 180,E1 -17365.606,E2 -17365.606} C_VEL
LIN {X 0,Y 275.284,Z 549.17,A -85,B 0,C 180,E1 -17367.073,E2 -17367.073} C_VEL
LIN {X 0,Y 275.29,Z 549.251,A -85,B 0,C 180,E1 -17368.537,E2 -17368.537} C_VEL
LIN {X 0,Y 275.331,Z 548.946,A -85,B 0,C 180,E1 -17369.999,E2 -17369.999} C_VEL
LIN {X 0,Y 275.314,Z 548.25,A -85,B 0,C 180,E1 -17371.462,E2 -17371.462} C_VEL
LIN {X 0,Y 275.329,Z 547.126,A -85,B 0,C 180,E1 -17372.926,E2 -17372.926} C_VEL
LIN {X 0,Y 275.36,Z 544.102,A -85,B 0,C 180,E1 -17375.496,E2 -17375.496} C_VEL
LIN {X 0,Y 275.589,Z 539.696,A -85,B 0,C 180,E1 -17378.062,E2 -17378.062} C_VEL
LIN {X 0,Y 276.027,Z 534.673,A -85,B 0,C 180,E1 -17380.266,E2 -17380.266} C_VEL
LIN {X 0,Y 276.767,Z 528.348,A -85,B 0,C 180,E1 -17382.464,E2 -17382.464} C_VEL
LIN {X 0,Y 277.885,Z 520.417,A -85,B 0,C 180,E1 -17384.649,E2 -17384.649} C_VEL
LIN {X 0,Y 279.212,Z 511.661,A -85,B 0,C 180,E1 -17386.587,E2 -17386.587} C_VEL
LIN {X 0,Y 280.487,Z 501.315,A -85,B 0,C 180,E1 -17388.441,E2 -17388.441} C_VEL
LIN {X 0,Y 282.095,Z 489.901,A -85,B 0,C 180,E1 -17390.032,E2 -17390.032} C_VEL
LIN {X 0,Y 283.499,Z 478.698,A -85,B 0,C 180,E1 -17391.257,E2 -17391.257} C_VEL
LIN {X 0,Y 284.791,Z 466.196,A -85,B 0,C 180,E1 -17392.297,E2 -17392.297} C_VEL
LIN {X 0,Y 285.884,Z 452.841,A -85,B 0,C 180,E1 -17393.066,E2 -17393.066} C_VEL
LIN {X 0,Y 286.42,Z 441.175,A -85,B 0,C 180,E1 -17393.501,E2 -17393.501} C_VEL
LIN {X 0,Y 287.75,Z 381.725,A -85,B 0,C 180,E1 -17394.974,E2 -17394.974} C_VEL
LIN {X 0,Y 282.372,Z 341.216,A -85,B 0,C 180,E1 -17396.485,E2 -17396.485} C_VEL
LIN {X 0,Y 281.435,Z 336.401,A -85,B 0,C 180,E1 -17396.711,E2 -17396.711} C_VEL
LIN {X 0,Y 279.345,Z 325.354,A -85,B 0,C 180,E1 -17400.21,E2 -17400.21} C_VEL
LIN {X 0,Y 277.261,Z 315.95,A -85,B 0,C 180,E1 -17403.398,E2 -17403.398} C_VEL
LIN {X 0,Y 277.306,Z 315.944,A -85,B 0,C 180,E1 -17405.805,E2 -17405.805} C_VEL
LIN {X 0,Y 277.236,Z 315.95,A -85,B 0,C 180,E1 -17409.327,E2 -17409.327} C_VEL
LIN {X 0,Y 277.208,Z 315.953,A -85,B 0,C 180,E1 -17413.197,E2 -17413.197} C_VEL
LIN {X 0,Y 277.213,Z 315.953,A -85,B 0,C 180,E1 -17417.324,E2 -17417.324} C_VEL
LIN {X 0,Y 277.259,Z 315.947,A -85,B 0,C 180,E1 -17421.792,E2 -17421.792} C_VEL
LIN {X 0,Y 277.281,Z 315.947,A -85,B 0,C 180,E1 -17424.341,E2 -17424.341} C_VEL
LIN {X 0,Y 277.241,Z 315.949,A -85,B 0,C 180,E1 -17427.836,E2 -17427.836} C_VEL
LIN {X 0,Y 277.283,Z 315.946,A -85,B 0,C 180,E1 -17431.211,E2 -17431.211} C_VEL
LIN {X 0,Y 277.308,Z 315.941,A -85,B 0,C 180,E1 -17434.479,E2 -17434.479} C_VEL
LIN {X 0,Y 277.282,Z 315.943,A -85,B 0,C 180,E1 -17437.654,E2 -17437.654} C_VEL
LIN {X 0,Y 277.342,Z 315.937,A -85,B 0,C 180,E1 -17440.766,E2 -17440.766} C_VEL
LIN {X 0,Y 277.431,Z 315.927,A -85,B 0,C 180,E1 -17445.325,E2 -17445.325} C_VEL
LIN {X 0,Y 277.503,Z 315.912,A -85,B 0,C 180,E1 -17449.788,E2 -17449.788} C_VEL
LIN {X 0,Y 277.645,Z 315.897,A -85,B 0,C 180,E1 -17452.729,E2 -17452.729} C_VEL
LIN {X 0,Y 277.817,Z 315.867,A -85,B 0,C 180,E1 -17458.55,E2 -17458.55} C_VEL
LIN {X 0,Y 277.816,Z 315.873,A -85,B 0,C 180,E1 -17461.449,E2 -17461.449} C_VEL
LIN {X 0,Y 277.607,Z 315.901,A -85,B 0,C 180,E1 -17467.272,E2 -17467.272} C_VEL
LIN {X 0,Y 277.455,Z 315.915,A -85,B 0,C 180,E1 -17470.213,E2 -17470.213} C_VEL
LIN {X 0,Y 277.43,Z 315.926,A -85,B 0,C 180,E1 -17474.674,E2 -17474.674} C_VEL
LIN {X 0,Y 277.338,Z 315.929,A -85,B 0,C 180,E1 -17479.234,E2 -17479.234} C_VEL
LIN {X 0,Y 277.288,Z 315.944,A -85,B 0,C 180,E1 -17484.158,E2 -17484.158} C_VEL
LIN {X 0,Y 277.322,Z 315.936,A -85,B 0,C 180,E1 -17487.505,E2 -17487.505} C_VEL
LIN {X 0,Y 277.268,Z 315.938,A -85,B 0,C 180,E1 -17490.482,E2 -17490.482} C_VEL
LIN {X 0,Y 277.243,Z 315.947,A -85,B 0,C 180,E1 -17493.896,E2 -17493.896} C_VEL
LIN {X 0,Y 277.26,Z 315.94,A -85,B 0,C 180,E1 -17497.47,E2 -17497.47} C_VEL
LIN {X 0,Y 277.205,Z 315.953,A -85,B 0,C 180,E1 -17501.237,E2 -17501.237} C_VEL
LIN {X 0,Y 277.19,Z 315.95,A -85,B 0,C 180,E1 -17505.228,E2 -17505.228} C_VEL
LIN {X 0,Y 277.193,Z 315.955,A -85,B 0,C 180,E1 -17509.519,E2 -17509.519} C_VEL
LIN {X 0,Y 277.257,Z 315.943,A -85,B 0,C 180,E1 -17512.53,E2 -17512.53} C_VEL
LIN {X 0,Y 277.243,Z 315.948,A -85,B 0,C 180,E1 -17516.105,E2 -17516.105} C_VEL
LIN {X 0,Y 277.225,Z 315.95,A -85,B 0,C 180,E1 -17519.535,E2 -17519.535} C_VEL
LIN {X 0,Y 277.251,Z 315.946,A -85,B 0,C 180,E1 -17522.854,E2 -17522.854} C_VEL
LIN {X 0,Y 277.269,Z 315.946,A -85,B 0,C 180,E1 -17526.075,E2 -17526.075} C_VEL
LIN {X 0,Y 277.323,Z 315.94,A -85,B 0,C 180,E1 -17530.765,E2 -17530.765} C_VEL
LIN {X 0,Y 277.366,Z 316.063,A -85,B 0,C 180,E1 -17532.47,E2 -17532.47} C_VEL
LIN {X 0,Y 277.791,Z 317.9,A -85,B 0,C 180,E1 -17533.07,E2 -17533.07} C_VEL
LIN {X 0,Y 285.719,Z 338.761,A -85,B 0,C 180,E1 -17534.315,E2 -17534.315} C_VEL
LIN {X 0,Y 287.882,Z 345.751,A -85,B 0,C 180,E1 -17534.676,E2 -17534.676} C_VEL
LIN {X 0,Y 288.521,Z 351.03,A -85,B 0,C 180,E1 -17534.866,E2 -17534.866} C_VEL
LIN {X 0,Y 286.626,Z 425.19,A -85,B 0,C 180,E1 -17536.711,E2 -17536.711} C_VEL
LIN {X 0,Y 285.968,Z 438.283,A -85,B 0,C 180,E1 -17537.312,E2 -17537.312} C_VEL
LIN {X 0,Y 285.091,Z 450.885,A -85,B 0,C 180,E1 -17538.176,E2 -17538.176} C_VEL
LIN {X 0,Y 283.943,Z 462.923,A -85,B 0,C 180,E1 -17539.302,E2 -17539.302} C_VEL
LIN {X 0,Y 282.224,Z 474.452,A -85,B 0,C 180,E1 -17540.685,E2 -17540.685} C_VEL
LIN {X 0,Y 280.953,Z 484.748,A -85,B 0,C 180,E1 -17542.273,E2 -17542.273} C_VEL
LIN {X 0,Y 279.663,Z 493.202,A -85,B 0,C 180,E1 -17543.869,E2 -17543.869} C_VEL
LIN {X 0,Y 278.383,Z 502.341,A -85,B 0,C 180,E1 -17546.02,E2 -17546.02} C_VEL
LIN {X 0,Y 277.216,Z 509.713,A -85,B 0,C 180,E1 -17548.185,E2 -17548.185} C_VEL
LIN {X 0,Y 276.364,Z 516.487,A -85,B 0,C 180,E1 -17550.729,E2 -17550.729} C_VEL
LIN {X 0,Y 275.781,Z 520.968,A -85,B 0,C 180,E1 -17552.922,E2 -17552.922} C_VEL
LIN {X 0,Y 275.684,Z 523.325,A -85,B 0,C 180,E1 -17554.387,E2 -17554.387} C_VEL
LIN {X 0,Y 275.582,Z 525.393,A -85,B 0,C 180,E1 -17555.963,E2 -17555.963} C_VEL
LIN {X 0,Y 275.327,Z 526.792,A -85,B 0,C 180,E1 -17557.333,E2 -17557.333} C_VEL
LIN {X 0,Y 275.212,Z 527.864,A -85,B 0,C 180,E1 -17558.814,E2 -17558.814} C_VEL
LIN {X 0,Y 275.245,Z 528.834,A -85,B 0,C 180,E1 -17561.787,E2 -17561.787} C_VEL
LIN {X 0,Y 275.586,Z 528.4,A -85,B 0,C 180,E1 -17564.287,E2 -17564.287} C_VEL
LIN {X 0,Y 275.94,Z 527.213,A -85,B 0,C 180,E1 -17566.27,E2 -17566.27} C_VEL
LIN {X 0,Y 276.315,Z 525.86,A -85,B 0,C 180,E1 -17567.772,E2 -17567.772} C_VEL
LIN {X 0,Y 277.329,Z 522.451,A -85,B 0,C 180,E1 -17570.341,E2 -17570.341} C_VEL
LIN {X 0,Y 278.775,Z 517.374,A -85,B 0,C 180,E1 -17573.002,E2 -17573.002} C_VEL
LIN {X 0,Y 280.343,Z 511.756,A -85,B 0,C 180,E1 -17575.226,E2 -17575.226} C_VEL
LIN {X 0,Y 282.258,Z 504.679,A -85,B 0,C 180,E1 -17577.428,E2 -17577.428} C_VEL
LIN {X 0,Y 284.568,Z 495.732,A -85,B 0,C 180,E1 -17579.6,E2 -17579.6} C_VEL
LIN {X 0,Y 286.798,Z 486.515,A -85,B 0,C 180,E1 -17581.382,E2 -17581.382} C_VEL
LIN {X 0,Y 288.94,Z 476.246,A -85,B 0,C 180,E1 -17582.973,E2 -17582.973} C_VEL
LIN {X 0,Y 290.897,Z 465.378,A -85,B 0,C 180,E1 -17584.301,E2 -17584.301} C_VEL
LIN {X 0,Y 292.709,Z 452.71,A -85,B 0,C 180,E1 -17585.503,E2 -17585.503} C_VEL
LIN {X 0,Y 293.929,Z 441.646,A -85,B 0,C 180,E1 -17586.284,E2 -17586.284} C_VEL
LIN {X 0,Y 294.797,Z 428.905,A -85,B 0,C 180,E1 -17586.924,E2 -17586.924} C_VEL
LIN {X 0,Y 295.706,Z 411.81,A -85,B 0,C 180,E1 -17587.386,E2 -17587.386} C_VEL
LIN {X 0,Y 297.604,Z 358.016,A -85,B 0,C 180,E1 -17588.669,E2 -17588.669} C_VEL
LIN {X 0,Y 291.151,Z 343.487,A -85,B 0,C 180,E1 -17589.915,E2 -17589.915} C_VEL
LIN {X 0,Y 283.961,Z 329.461,A -85,B 0,C 180,E1 -17591.329,E2 -17591.329} C_VEL
LIN {X 0,Y 279.448,Z 321.611,A -85,B 0,C 180,E1 -17592.24,E2 -17592.24} C_VEL
LIN {X 0,Y 277.873,Z 318.475,A -85,B 0,C 180,E1 -17592.62,E2 -17592.62} C_VEL
LIN {X 0,Y 277.219,Z 315.951,A -85,B 0,C 180,E1 -17593.715,E2 -17593.715} C_VEL
LIN {X 0,Y 277.215,Z 315.953,A -85,B 0,C 180,E1 -17597.325,E2 -17597.325} C_VEL
LIN {X 0,Y 277.261,Z 315.942,A -85,B 0,C 180,E1 -17601.794,E2 -17601.794} C_VEL
LIN {X 0,Y 277.283,Z 315.941,A -85,B 0,C 180,E1 -17604.342,E2 -17604.342} C_VEL
LIN {X 0,Y 277.227,Z 315.938,A -85,B 0,C 180,E1 -17608.544,E2 -17608.544} C_VEL
LIN {X 0,Y 277.359,Z 315.921,A -85,B 0,C 180,E1 -17612.864,E2 -17612.864} C_VEL
LIN {X 0,Y 277.289,Z 315.934,A -85,B 0,C 180,E1 -17614.848,E2 -17614.848} C_VEL
LIN {X 0,Y 276.597,Z 316.02,A -85,B 0,C 180,E1 -17616.061,E2 -17616.061} C_VEL
LIN {X 0,Y 273.746,Z 316.382,A -85,B 0,C 180,E1 -17618.037,E2 -17618.037} C_VEL
LIN {X 0,Y 271.354,Z 316.675,A -85,B 0,C 180,E1 -17619.643,E2 -17619.643} C_VEL
LIN {X 0,Y 270.344,Z 316.798,A -85,B 0,C 180,E1 -17620.887,E2 -17620.887} C_VEL
LIN {X 0,Y 270.269,Z 316.81,A -85,B 0,C 180,E1 -17621.308,E2 -17621.308} C_VEL
LIN {X 0,Y 270.403,Z 316.792,A -85,B 0,C 180,E1 -17624.936,E2 -17624.936} C_VEL
LIN {X 0,Y 270.442,Z 316.789,A -85,B 0,C 180,E1 -17629.519,E2 -17629.519} C_VEL
LIN {X 0,Y 270.611,Z 316.77,A -85,B 0,C 180,E1 -17632.539,E2 -17632.539} C_VEL
LIN {X 0,Y 270.787,Z 316.745,A -85,B 0,C 180,E1 -17638.513,E2 -17638.513} C_VEL
LIN {X 0,Y 270.787,Z 316.749,A -85,B 0,C 180,E1 -17641.488,E2 -17641.488} C_VEL
LIN {X 0,Y 270.612,Z 316.762,A -85,B 0,C 180,E1 -17647.461,E2 -17647.461} C_VEL
LIN {X 0,Y 270.443,Z 316.79,A -85,B 0,C 180,E1 -17650.481,E2 -17650.481} C_VEL
LIN {X 0,Y 270.404,Z 316.795,A -85,B 0,C 180,E1 -17655.065,E2 -17655.065} C_VEL
LIN {X 0,Y 270.303,Z 316.808,A -85,B 0,C 180,E1 -17659.756,E2 -17659.756} C_VEL
LIN {X 0,Y 270.24,Z 316.814,A -85,B 0,C 180,E1 -17664.589,E2 -17664.589} C_VEL
LIN {X 0,Y 270.272,Z 316.814,A -85,B 0,C 180,E1 -17667.909,E2 -17667.909} C_VEL
LIN {X 0,Y 270.186,Z 316.826,A -85,B 0,C 180,E1 -17671.348,E2 -17671.348} C_VEL
LIN {X 0,Y 270.204,Z 316.824,A -85,B 0,C 180,E1 -17674.906,E2 -17674.906} C_VEL
LIN {X 0,Y 270.199,Z 316.816,A -85,B 0,C 180,E1 -17678.711,E2 -17678.711} C_VEL
LIN {X 0,Y 270.173,Z 316.825,A -85,B 0,C 180,E1 -17682.558,E2 -17682.558} C_VEL
LIN {X 0,Y 270.167,Z 316.83,A -85,B 0,C 180,E1 -17686.751,E2 -17686.751} C_VEL
LIN {X 0,Y 270.224,Z 316.932,A -85,B 0,C 180,E1 -17689.682,E2 -17689.682} C_VEL
LIN {X 0,Y 272.843,Z 326.42,A -85,B 0,C 180,E1 -17693.669,E2 -17693.669} C_VEL
LIN {X 0,Y 275.017,Z 335.376,A -85,B 0,C 180,E1 -17697.052,E2 -17697.052} C_VEL
LIN {X 0,Y 283.089,Z 351.998,A -85,B 0,C 180,E1 -17698.77,E2 -17698.77} C_VEL
LIN {X 0,Y 285.875,Z 358.956,A -85,B 0,C 180,E1 -17699.367,E2 -17699.367} C_VEL
LIN {X 0,Y 289.841,Z 380.49,A -85,B 0,C 180,E1 -17700.53,E2 -17700.53} C_VEL
LIN {X 0,Y 290.735,Z 387.438,A -85,B 0,C 180,E1 -17700.846,E2 -17700.846} C_VEL
LIN {X 0,Y 288.588,Z 445.091,A -85,B 0,C 180,E1 -17702.292,E2 -17702.292} C_VEL
LIN {X 0,Y 287.355,Z 458.721,A -85,B 0,C 180,E1 -17702.901,E2 -17702.901} C_VEL
LIN {X 0,Y 285.707,Z 471.042,A -85,B 0,C 180,E1 -17703.719,E2 -17703.719} C_VEL
LIN {X 0,Y 283.832,Z 482.075,A -85,B 0,C 180,E1 -17704.714,E2 -17704.714} C_VEL
LIN {X 0,Y 281.501,Z 493.59,A -85,B 0,C 180,E1 -17706.065,E2 -17706.065} C_VEL
LIN {X 0,Y 279.166,Z 503.972,A -85,B 0,C 180,E1 -17707.618,E2 -17707.618} C_VEL
LIN {X 0,Y 277.043,Z 512.478,A -85,B 0,C 180,E1 -17709.197,E2 -17709.197} C_VEL
LIN {X 0,Y 274.802,Z 520.951,A -85,B 0,C 180,E1 -17711.133,E2 -17711.133} C_VEL
LIN {X 0,Y 272.738,Z 529.172,A -85,B 0,C 180,E1 -17713.533,E2 -17713.533} C_VEL
LIN {X 0,Y 271.02,Z 535.175,A -85,B 0,C 180,E1 -17715.738,E2 -17715.738} C_VEL
LIN {X 0,Y 269.778,Z 539.946,A -85,B 0,C 180,E1 -17717.97,E2 -17717.97} C_VEL
LIN {X 0,Y 268.972,Z 543.622,A -85,B 0,C 180,E1 -17720.221,E2 -17720.221} C_VEL
LIN {X 0,Y 268.421,Z 546.303,A -85,B 0,C 180,E1 -17722.477,E2 -17722.477} C_VEL
LIN {X 0,Y 268.165,Z 548.464,A -85,B 0,C 180,E1 -17725.49,E2 -17725.49} C_VEL
LIN {X 0,Y 268.194,Z 548.915,A -85,B 0,C 180,E1 -17726.995,E2 -17726.995} C_VEL
LIN {X 0,Y 268.215,Z 548.976,A -85,B 0,C 180,E1 -17728.498,E2 -17728.498} C_VEL
LIN {X 0,Y 268.252,Z 548.651,A -85,B 0,C 180,E1 -17729.999,E2 -17729.999} C_VEL
LIN {X 0,Y 268.239,Z 547.931,A -85,B 0,C 180,E1 -17731.501,E2 -17731.501} C_VEL
LIN {X 0,Y 268.237,Z 546.766,A -85,B 0,C 180,E1 -17733.003,E2 -17733.003} C_VEL
LIN {X 0,Y 268.254,Z 544.048,A -85,B 0,C 180,E1 -17735.395,E2 -17735.395} C_VEL
LIN {X 0,Y 268.426,Z 540.683,A -85,B 0,C 180,E1 -17737.522,E2 -17737.522} C_VEL
LIN {X 0,Y 268.809,Z 535.999,A -85,B 0,C 180,E1 -17739.784,E2 -17739.784} C_VEL
LIN {X 0,Y 269.634,Z 528.916,A -85,B 0,C 180,E1 -17742.417,E2 -17742.417} C_VEL
LIN {X 0,Y 270.787,Z 521.244,A -85,B 0,C 180,E1 -17744.657,E2 -17744.657} C_VEL
LIN {X 0,Y 272.226,Z 511.818,A -85,B 0,C 180,E1 -17746.832,E2 -17746.832} C_VEL
LIN {X 0,Y 273.548,Z 501.562,A -85,B 0,C 180,E1 -17748.732,E2 -17748.732} C_VEL
LIN {X 0,Y 275.197,Z 490.315,A -85,B 0,C 180,E1 -17750.362,E2 -17750.362} C_VEL
LIN {X 0,Y 276.641,Z 479.274,A -85,B 0,C 180,E1 -17751.614,E2 -17751.614} C_VEL
LIN {X 0,Y 277.976,Z 467.041,A -85,B 0,C 180,E1 -17752.678,E2 -17752.678} C_VEL
LIN {X 0,Y 279.063,Z 454.3,A -85,B 0,C 180,E1 -17753.467,E2 -17753.467} C_VEL
LIN {X 0,Y 279.742,Z 441.313,A -85,B 0,C 180,E1 -17753.98,E2 -17753.98} C_VEL
LIN {X 0,Y 281.197,Z 383.515,A -85,B 0,C 180,E1 -17755.438,E2 -17755.438} C_VEL
LIN {X 0,Y 276.395,Z 345.997,A -85,B 0,C 180,E1 -17756.863,E2 -17756.863} C_VEL
LIN {X 0,Y 275.086,Z 338.861,A -85,B 0,C 180,E1 -17757.176,E2 -17757.176} C_VEL
LIN {X 0,Y 274.22,Z 336.035,A -85,B 0,C 180,E1 -17757.372,E2 -17757.372} C_VEL
LIN {X 0,Y 272.214,Z 326.01,A -85,B 0,C 180,E1 -17760.657,E2 -17760.657} C_VEL
LIN {X 0,Y 270.228,Z 316.826,A -85,B 0,C 180,E1 -17763.875,E2 -17763.875} C_VEL
LIN {X 0,Y 270.227,Z 316.824,A -85,B 0,C 180,E1 -17766.738,E2 -17766.738} C_VEL
LIN {X 0,Y 270.168,Z 316.831,A -85,B 0,C 180,E1 -17771.027,E2 -17771.027} C_VEL
LIN {X 0,Y 270.151,Z 316.832,A -85,B 0,C 180,E1 -17775.379,E2 -17775.379} C_VEL
LIN {X 0,Y 270.172,Z 316.83,A -85,B 0,C 180,E1 -17779.433,E2 -17779.433} C_VEL
LIN {X 0,Y 270.223,Z 316.824,A -85,B 0,C 180,E1 -17783.73,E2 -17783.73} C_VEL
LIN {X 0,Y 270.2,Z 316.831,A -85,B 0,C 180,E1 -17786.892,E2 -17786.892} C_VEL
LIN {X 0,Y 270.225,Z 316.825,A -85,B 0,C 180,E1 -17790.386,E2 -17790.386} C_VEL
LIN {X 0,Y 270.258,Z 316.819,A -85,B 0,C 180,E1 -17793.763,E2 -17793.763} C_VEL
LIN {X 0,Y 270.23,Z 316.827,A -85,B 0,C 180,E1 -17797.038,E2 -17797.038} C_VEL
LIN {X 0,Y 270.299,Z 316.813,A -85,B 0,C 180,E1 -17800.244,E2 -17800.244} C_VEL
LIN {X 0,Y 270.399,Z 316.802,A -85,B 0,C 180,E1 -17804.935,E2 -17804.935} C_VEL
LIN {X 0,Y 270.438,Z 316.788,A -85,B 0,C 180,E1 -17809.518,E2 -17809.518} C_VEL
LIN {X 0,Y 270.604,Z 316.774,A -85,B 0,C 180,E1 -17812.538,E2 -17812.538} C_VEL
LIN {X 0,Y 270.783,Z 316.742,A -85,B 0,C 180,E1 -17818.512,E2 -17818.512} C_VEL
LIN {X 0,Y 270.782,Z 316.749,A -85,B 0,C 180,E1 -17821.487,E2 -17821.487} C_VEL
LIN {X 0,Y 270.567,Z 316.778,A -85,B 0,C 180,E1 -17827.462,E2 -17827.462} C_VEL
LIN {X 0,Y 270.408,Z 316.793,A -85,B 0,C 180,E1 -17830.482,E2 -17830.482} C_VEL
LIN {X 0,Y 270.398,Z 316.8,A -85,B 0,C 180,E1 -17835.065,E2 -17835.065} C_VEL
LIN {X 0,Y 270.295,Z 316.806,A -85,B 0,C 180,E1 -17839.756,E2 -17839.756} C_VEL
LIN {X 0,Y 270.234,Z 316.825,A -85,B 0,C 180,E1 -17844.589,E2 -17844.589} C_VEL
LIN {X 0,Y 270.268,Z 316.815,A -85,B 0,C 180,E1 -17847.909,E2 -17847.909} C_VEL
LIN {X 0,Y 270.18,Z 316.822,A -85,B 0,C 180,E1 -17851.348,E2 -17851.348} C_VEL
LIN {X 0,Y 270.197,Z 316.827,A -85,B 0,C 180,E1 -17854.906,E2 -17854.906} C_VEL
LIN {X 0,Y 270.193,Z 316.82,A -85,B 0,C 180,E1 -17858.711,E2 -17858.711} C_VEL
LIN {X 0,Y 270.168,Z 316.83,A -85,B 0,C 180,E1 -17862.559,E2 -17862.559} C_VEL
LIN {X 0,Y 270.144,Z 316.828,A -85,B 0,C 180,E1 -17866.755,E2 -17866.755} C_VEL
LIN {X 0,Y 270.204,Z 316.823,A -85,B 0,C 180,E1 -17871.375,E2 -17871.375} C_VEL
LIN {X 0,Y 270.198,Z 316.83,A -85,B 0,C 180,E1 -17875.095,E2 -17875.095} C_VEL
LIN {X 0,Y 270.168,Z 316.832,A -85,B 0,C 180,E1 -17879.142,E2 -17879.142} C_VEL
LIN {X 0,Y 270.186,Z 316.825,A -85,B 0,C 180,E1 -17882.177,E2 -17882.177} C_VEL
LIN {X 0,Y 270.214,Z 316.827,A -85,B 0,C 180,E1 -17885.548,E2 -17885.548} C_VEL
LIN {X 0,Y 270.259,Z 316.821,A -85,B 0,C 180,E1 -17890.242,E2 -17890.242} C_VEL
LIN {X 0,Y 270.286,Z 316.888,A -85,B 0,C 180,E1 -17891.996,E2 -17891.996} C_VEL
LIN {X 0,Y 270.648,Z 318.309,A -85,B 0,C 180,E1 -17892.427,E2 -17892.427} C_VEL
LIN {X 0,Y 278.575,Z 338.607,A -85,B 0,C 180,E1 -17893.711,E2 -17893.711} C_VEL
LIN {X 0,Y 281.521,Z 348.011,A -85,B 0,C 180,E1 -17894.218,E2 -17894.218} C_VEL
LIN {X 0,Y 281.924,Z 351.983,A -85,B 0,C 180,E1 -17894.359,E2 -17894.359} C_VEL
LIN {X 0,Y 279.936,Z 426.044,A -85,B 0,C 180,E1 -17896.249,E2 -17896.249} C_VEL
LIN {X 0,Y 279.215,Z 439.695,A -85,B 0,C 180,E1 -17896.907,E2 -17896.907} C_VEL
LIN {X 0,Y 278.304,Z 451.983,A -85,B 0,C 180,E1 -17897.791,E2 -17897.791} C_VEL
LIN {X 0,Y 277.043,Z 464.57,A -85,B 0,C 180,E1 -17899.033,E2 -17899.033} C_VEL
LIN {X 0,Y 275.433,Z 474.566,A -85,B 0,C 180,E1 -17900.268,E2 -17900.268} C_VEL
LIN {X 0,Y 274.103,Z 484.889,A -85,B 0,C 180,E1 -17901.894,E2 -17901.894} C_VEL
LIN {X 0,Y 272.632,Z 494.214,A -85,B 0,C 180,E1 -17903.711,E2 -17903.711} C_VEL
LIN {X 0,Y 271.321,Z 503.201,A -85,B 0,C 180,E1 -17905.916,E2 -17905.916} C_VEL
LIN {X 0,Y 270.115,Z 510.471,A -85,B 0,C 180,E1 -17908.137,E2 -17908.137} C_VEL
LIN {X 0,Y 269.481,Z 515.379,A -85,B 0,C 180,E1 -17910.001,E2 -17910.001} C_VEL
LIN {X 0,Y 268.836,Z 520.162,A -85,B 0,C 180,E1 -17912.248,E2 -17912.248} C_VEL
LIN {X 0,Y 268.584,Z 523.825,A -85,B 0,C 180,E1 -17914.503,E2 -17914.503} C_VEL
LIN {X 0,Y 268.48,Z 525.725,A -85,B 0,C 180,E1 -17916.011,E2 -17916.011} C_VEL
LIN {X 0,Y 268.225,Z 527.186,A -85,B 0,C 180,E1 -17917.528,E2 -17917.528} C_VEL
LIN {X 0,Y 268.103,Z 528.22,A -85,B 0,C 180,E1 -17919.05,E2 -17919.05} C_VEL
LIN {X 0,Y 268.19,Z 529.118,A -85,B 0,C 180,E1 -17922.102,E2 -17922.102} C_VEL
LIN {X 0,Y 268.512,Z 528.687,A -85,B 0,C 180,E1 -17924.435,E2 -17924.435} C_VEL
LIN {X 0,Y 268.949,Z 527.356,A -85,B 0,C 180,E1 -17926.705,E2 -17926.705} C_VEL
LIN {X 0,Y 269.373,Z 525.95,A -85,B 0,C 180,E1 -17928.245,E2 -17928.245} C_VEL
LIN {X 0,Y 270.372,Z 522.82,A -85,B 0,C 180,E1 -17930.647,E2 -17930.647} C_VEL
LIN {X 0,Y 271.578,Z 518.914,A -85,B 0,C 180,E1 -17932.841,E2 -17932.841} C_VEL
LIN {X 0,Y 273.437,Z 512.597,A -85,B 0,C 180,E1 -17935.501,E2 -17935.501} C_VEL
LIN {X 0,Y 275.421,Z 505.668,A -85,B 0,C 180,E1 -17937.755,E2 -17937.755} C_VEL
LIN {X 0,Y 277.369,Z 498.546,A -85,B 0,C 180,E1 -17939.61,E2 -17939.61} C_VEL
LIN {X 0,Y 279.817,Z 489.087,A -85,B 0,C 180,E1 -17941.583,E2 -17941.583} C_VEL
LIN {X 0,Y 282.077,Z 479.125,A -85,B 0,C 180,E1 -17943.239,E2 -17943.239} C_VEL
LIN {X 0,Y 284.161,Z 468.364,A -85,B 0,C 180,E1 -17944.67,E2 -17944.67} C_VEL
LIN {X 0,Y 285.957,Z 457.492,A -85,B 0,C 180,E1 -17945.802,E2 -17945.802} C_VEL
LIN {X 0,Y 287.476,Z 444.942,A -85,B 0,C 180,E1 -17946.795,E2 -17946.795} C_VEL
LIN {X 0,Y 288.582,Z 431.607,A -85,B 0,C 180,E1 -17947.542,E2 -17947.542} C_VEL
LIN {X 0,Y 289.422,Z 418.584,A -85,B 0,C 180,E1 -17947.955,E2 -17947.955} C_VEL
LIN {X 0,Y 291.539,Z 359.894,A -85,B 0,C 180,E1 -17949.384,E2 -17949.384} C_VEL
LIN {X 0,Y 285.519,Z 346.389,A -85,B 0,C 180,E1 -17950.594,E2 -17950.594} C_VEL
LIN {X 0,Y 279.074,Z 333.746,A -85,B 0,C 180,E1 -17951.915,E2 -17951.915} C_VEL
LIN {X 0,Y 272.407,Z 322.129,A -85,B 0,C 180,E1 -17953.326,E2 -17953.326} C_VEL
LIN {X 0,Y 270.716,Z 318.832,A -85,B 0,C 180,E1 -17953.748,E2 -17953.748} C_VEL
LIN {X 0,Y 270.159,Z 316.829,A -85,B 0,C 180,E1 -17954.684,E2 -17954.684} C_VEL
LIN {X 0,Y 270.169,Z 316.83,A -85,B 0,C 180,E1 -17958.972,E2 -17958.972} C_VEL
LIN {X 0,Y 270.216,Z 316.82,A -85,B 0,C 180,E1 -17963.259,E2 -17963.259} C_VEL
LIN {X 0,Y 270.203,Z 316.82,A -85,B 0,C 180,E1 -17966.893,E2 -17966.893} C_VEL
LIN {X 0,Y 270.229,Z 316.815,A -85,B 0,C 180,E1 -17970.387,E2 -17970.387} C_VEL
LIN {X 0,Y 270.262,Z 316.811,A -85,B 0,C 180,E1 -17973.764,E2 -17973.764} C_VEL
LIN {X 0,Y 270.21,Z 316.813,A -85,B 0,C 180,E1 -17977.037,E2 -17977.037} C_VEL
LIN {X 0,Y 270.3,Z 316.803,A -85,B 0,C 180,E1 -17980.245,E2 -17980.245} C_VEL
LIN {X 0,Y 270.269,Z 316.81,A -85,B 0,C 180,E1 -17981.308,E2 -17981.308} C_VEL
LIN {X 0,Y 269.634,Z 316.899,A -85,B 0,C 180,E1 -17982.552,E2 -17982.552} C_VEL
LIN {X 0,Y 266.838,Z 317.256,A -85,B 0,C 180,E1 -17984.581,E2 -17984.581} C_VEL
LIN {X 0,Y 264.448,Z 317.551,A -85,B 0,C 180,E1 -17986.23,E2 -17986.23} C_VEL
LIN {X 0,Y 263.417,Z 317.672,A -85,B 0,C 180,E1 -17987.507,E2 -17987.507} C_VEL
LIN {X 0,Y 263.33,Z 317.678,A -85,B 0,C 180,E1 -17987.94,E2 -17987.94} C_VEL
LIN {X 0,Y 263.56,Z 317.653,A -85,B 0,C 180,E1 -17990.794,E2 -17990.794} C_VEL
LIN {X 0,Y 263.515,Z 317.651,A -85,B 0,C 180,E1 -17993.876,E2 -17993.876} C_VEL
LIN {X 0,Y 263.751,Z 317.621,A -85,B 0,C 180,E1 -17998.473,E2 -17998.473} C_VEL
LIN {X 0,Y 263.751,Z 317.624,A -85,B 0,C 180,E1 -18001.527,E2 -18001.527} C_VEL
LIN {X 0,Y 263.573,Z 317.639,A -85,B 0,C 180,E1 -18007.662,E2 -18007.662} C_VEL
LIN {X 0,Y 263.375,Z 317.668,A -85,B 0,C 180,E1 -18010.766,E2 -18010.766} C_VEL
LIN {X 0,Y 263.352,Z 317.671,A -85,B 0,C 180,E1 -18015.478,E2 -18015.478} C_VEL
LIN {X 0,Y 263.264,Z 317.681,A -85,B 0,C 180,E1 -18020.307,E2 -18020.307} C_VEL
LIN {X 0,Y 263.195,Z 317.693,A -85,B 0,C 180,E1 -18025.293,E2 -18025.293} C_VEL
LIN {X 0,Y 263.168,Z 317.695,A -85,B 0,C 180,E1 -18028.731,E2 -18028.731} C_VEL
LIN {X 0,Y 263.135,Z 317.7,A -85,B 0,C 180,E1 -18032.288,E2 -18032.288} C_VEL
LIN {X 0,Y 263.185,Z 317.696,A -85,B 0,C 180,E1 -18036.764,E2 -18036.764} C_VEL
LIN {X 0,Y 263.126,Z 317.687,A -85,B 0,C 180,E1 -18041.594,E2 -18041.594} C_VEL
LIN {X 0,Y 263.126,Z 317.709,A -85,B 0,C 180,E1 -18046.151,E2 -18046.151} C_VEL
LIN {X 0,Y 263.154,Z 317.854,A -85,B 0,C 180,E1 -18048.672,E2 -18048.672} C_VEL
LIN {X 0,Y 265.908,Z 327.524,A -85,B 0,C 180,E1 -18052.926,E2 -18052.926} C_VEL
LIN {X 0,Y 267.661,Z 334.837,A -85,B 0,C 180,E1 -18055.849,E2 -18055.849} C_VEL
LIN {X 0,Y 269.935,Z 339.274,A -85,B 0,C 180,E1 -18056.372,E2 -18056.372} C_VEL
LIN {X 0,Y 276.605,Z 352.949,A -85,B 0,C 180,E1 -18057.854,E2 -18057.854} C_VEL
LIN {X 0,Y 280.299,Z 361.707,A -85,B 0,C 180,E1 -18058.67,E2 -18058.67} C_VEL
LIN {X 0,Y 284.064,Z 382.797,A -85,B 0,C 180,E1 -18059.836,E2 -18059.836} C_VEL
LIN {X 0,Y 284.736,Z 388.908,A -85,B 0,C 180,E1 -18060.109,E2 -18060.109} C_VEL
LIN {X 0,Y 282.552,Z 444.613,A -85,B 0,C 180,E1 -18061.526,E2 -18061.526} C_VEL
LIN {X 0,Y 281.349,Z 457.845,A -85,B 0,C 180,E1 -18062.122,E2 -18062.122} C_VEL
LIN {X 0,Y 279.556,Z 470.877,A -85,B 0,C 180,E1 -18062.993,E2 -18062.993} C_VEL
LIN {X 0,Y 277.461,Z 482.671,A -85,B 0,C 180,E1 -18064.091,E2 -18064.091} C_VEL
LIN {X 0,Y 275.04,Z 494.03,A -85,B 0,C 180,E1 -18065.466,E2 -18065.466} C_VEL
LIN {X 0,Y 272.636,Z 504.289,A -85,B 0,C 180,E1 -18067.052,E2 -18067.052} C_VEL
LIN {X 0,Y 270.413,Z 512.697,A -85,B 0,C 180,E1 -18068.662,E2 -18068.662} C_VEL
LIN {X 0,Y 267.962,Z 521.521,A -85,B 0,C 180,E1 -18070.77,E2 -18070.77} C_VEL
LIN {X 0,Y 265.912,Z 529.212,A -85,B 0,C 180,E1 -18073.098,E2 -18073.098} C_VEL
LIN {X 0,Y 264.138,Z 535.157,A -85,B 0,C 180,E1 -18075.358,E2 -18075.358} C_VEL
LIN {X 0,Y 262.791,Z 539.873,A -85,B 0,C 180,E1 -18077.646,E2 -18077.646} C_VEL
LIN {X 0,Y 261.951,Z 543.5,A -85,B 0,C 180,E1 -18079.956,E2 -18079.956} C_VEL
LIN {X 0,Y 261.356,Z 546.134,A -85,B 0,C 180,E1 -18082.273,E2 -18082.273} C_VEL
LIN {X 0,Y 261.086,Z 547.989,A -85,B 0,C 180,E1 -18084.864,E2 -18084.864} C_VEL
LIN {X 0,Y 261.106,Z 548.661,A -85,B 0,C 180,E1 -18086.914,E2 -18086.914} C_VEL
LIN {X 0,Y 261.141,Z 548.702,A -85,B 0,C 180,E1 -18088.457,E2 -18088.457} C_VEL
LIN {X 0,Y 261.176,Z 548.355,A -85,B 0,C 180,E1 -18089.999,E2 -18089.999} C_VEL
LIN {X 0,Y 261.164,Z 547.604,A -85,B 0,C 180,E1 -18091.541,E2 -18091.541} C_VEL
LIN {X 0,Y 261.148,Z 546.405,A -85,B 0,C 180,E1 -18093.085,E2 -18093.085} C_VEL
LIN {X 0,Y 261.158,Z 543.966,A -85,B 0,C 180,E1 -18095.308,E2 -18095.308} C_VEL
LIN {X 0,Y 261.354,Z 540.228,A -85,B 0,C 180,E1 -18097.726,E2 -18097.726} C_VEL
LIN {X 0,Y 261.76,Z 535.491,A -85,B 0,C 180,E1 -18100.05,E2 -18100.05} C_VEL
LIN {X 0,Y 262.666,Z 528.352,A -85,B 0,C 180,E1 -18102.752,E2 -18102.752} C_VEL
LIN {X 0,Y 263.846,Z 520.593,A -85,B 0,C 180,E1 -18105.052,E2 -18105.052} C_VEL
LIN {X 0,Y 265.305,Z 511.532,A -85,B 0,C 180,E1 -18107.183,E2 -18107.183} C_VEL
LIN {X 0,Y 266.616,Z 501.798,A -85,B 0,C 180,E1 -18109.038,E2 -18109.038} C_VEL
LIN {X 0,Y 268.308,Z 490.712,A -85,B 0,C 180,E1 -18110.708,E2 -18110.708} C_VEL
LIN {X 0,Y 269.793,Z 479.826,A -85,B 0,C 180,E1 -18111.99,E2 -18111.99} C_VEL
LIN {X 0,Y 271.149,Z 467.813,A -85,B 0,C 180,E1 -18113.08,E2 -18113.08} C_VEL
LIN {X 0,Y 272.361,Z 454.79,A -85,B 0,C 180,E1 -18113.928,E2 -18113.928} C_VEL
LIN {X 0,Y 273.072,Z 441.945,A -85,B 0,C 180,E1 -18114.464,E2 -18114.464} C_VEL
LIN {X 0,Y 274.573,Z 383.894,A -85,B 0,C 180,E1 -18115.967,E2 -18115.967} C_VEL
LIN {X 0,Y 269.659,Z 345.544,A -85,B 0,C 180,E1 -18117.476,E2 -18117.476} C_VEL
LIN {X 0,Y 268.713,Z 341.005,A -85,B 0,C 180,E1 -18117.693,E2 -18117.693} C_VEL
LIN {X 0,Y 266.996,Z 335.79,A -85,B 0,C 180,E1 -18118.034,E2 -18118.034} C_VEL
LIN {X 0,Y 264.848,Z 325.405,A -85,B 0,C 180,E1 -18121.56,E2 -18121.56} C_VEL
LIN {X 0,Y 263.16,Z 317.706,A -85,B 0,C 180,E1 -18124.32,E2 -18124.32} C_VEL
LIN {X 0,Y 263.162,Z 317.704,A -85,B 0,C 180,E1 -18127.895,E2 -18127.895} C_VEL
LIN {X 0,Y 263.122,Z 317.709,A -85,B 0,C 180,E1 -18131.892,E2 -18131.892} C_VEL
LIN {X 0,Y 263.103,Z 317.712,A -85,B 0,C 180,E1 -18136.154,E2 -18136.154} C_VEL
LIN {X 0,Y 263.103,Z 317.711,A -85,B 0,C 180,E1 -18140.127,E2 -18140.127} C_VEL
LIN {X 0,Y 263.16,Z 317.705,A -85,B 0,C 180,E1 -18144.017,E2 -18144.017} C_VEL
LIN {X 0,Y 263.13,Z 317.707,A -85,B 0,C 180,E1 -18147.711,E2 -18147.711} C_VEL
LIN {X 0,Y 263.197,Z 317.698,A -85,B 0,C 180,E1 -18151.783,E2 -18151.783} C_VEL
LIN {X 0,Y 263.223,Z 317.698,A -85,B 0,C 180,E1 -18155.2,E2 -18155.2} C_VEL
LIN {X 0,Y 263.26,Z 317.691,A -85,B 0,C 180,E1 -18159.693,E2 -18159.693} C_VEL
LIN {X 0,Y 263.348,Z 317.679,A -85,B 0,C 180,E1 -18164.521,E2 -18164.521} C_VEL
LIN {X 0,Y 263.37,Z 317.666,A -85,B 0,C 180,E1 -18169.234,E2 -18169.234} C_VEL
LIN {X 0,Y 263.566,Z 317.651,A -85,B 0,C 180,E1 -18172.338,E2 -18172.338} C_VEL
LIN {X 0,Y 263.747,Z 317.618,A -85,B 0,C 180,E1 -18178.473,E2 -18178.473} C_VEL
LIN {X 0,Y 263.746,Z 317.625,A -85,B 0,C 180,E1 -18181.527,E2 -18181.527} C_VEL
LIN {X 0,Y 263.529,Z 317.655,A -85,B 0,C 180,E1 -18187.663,E2 -18187.663} C_VEL
LIN {X 0,Y 263.35,Z 317.67,A -85,B 0,C 180,E1 -18190.766,E2 -18190.766} C_VEL
LIN {X 0,Y 263.346,Z 317.68,A -85,B 0,C 180,E1 -18195.478,E2 -18195.478} C_VEL
LIN {X 0,Y 263.258,Z 317.681,A -85,B 0,C 180,E1 -18200.307,E2 -18200.307} C_VEL
LIN {X 0,Y 263.189,Z 317.699,A -85,B 0,C 180,E1 -18205.293,E2 -18205.293} C_VEL
LIN {X 0,Y 263.176,Z 317.694,A -85,B 0,C 180,E1 -18208.73,E2 -18208.73} C_VEL
LIN {X 0,Y 263.129,Z 317.702,A -85,B 0,C 180,E1 -18212.288,E2 -18212.288} C_VEL
LIN {X 0,Y 263.177,Z 317.698,A -85,B 0,C 180,E1 -18216.763,E2 -18216.763} C_VEL
LIN {X 0,Y 263.12,Z 317.706,A -85,B 0,C 180,E1 -18221.594,E2 -18221.594} C_VEL
LIN {X 0,Y 263.078,Z 317.704,A -85,B 0,C 180,E1 -18226.008,E2 -18226.008} C_VEL
LIN {X 0,Y 263.088,Z 317.711,A -85,B 0,C 180,E1 -18230.125,E2 -18230.125} C_VEL
LIN {X 0,Y 263.158,Z 317.703,A -85,B 0,C 180,E1 -18234.018,E2 -18234.018} C_VEL
LIN {X 0,Y 263.123,Z 317.708,A -85,B 0,C 180,E1 -18237.711,E2 -18237.711} C_VEL
LIN {X 0,Y 263.134,Z 317.705,A -85,B 0,C 180,E1 -18241.81,E2 -18241.81} C_VEL
LIN {X 0,Y 263.135,Z 317.706,A -85,B 0,C 180,E1 -18246.383,E2 -18246.383} C_VEL
LIN {X 0,Y 263.236,Z 317.697,A -85,B 0,C 180,E1 -18249.692,E2 -18249.692} C_VEL
LIN {X 0,Y 263.243,Z 317.817,A -85,B 0,C 180,E1 -18251.536,E2 -18251.536} C_VEL
LIN {X 0,Y 263.361,Z 318.466,A -85,B 0,C 180,E1 -18251.726,E2 -18251.726} C_VEL
LIN {X 0,Y 270.011,Z 334.983,A -85,B 0,C 180,E1 -18252.845,E2 -18252.845} C_VEL
LIN {X 0,Y 274.864,Z 348.848,A -85,B 0,C 180,E1 -18253.673,E2 -18253.673} C_VEL
LIN {X 0,Y 275.356,Z 352.636,A -85,B 0,C 180,E1 -18253.822,E2 -18253.822} C_VEL
LIN {X 0,Y 273.325,Z 425.699,A -85,B 0,C 180,E1 -18255.719,E2 -18255.719} C_VEL
LIN {X 0,Y 272.627,Z 438.794,A -85,B 0,C 180,E1 -18256.348,E2 -18256.348} C_VEL
LIN {X 0,Y 271.62,Z 451.961,A -85,B 0,C 180,E1 -18257.296,E2 -18257.296} C_VEL
LIN {X 0,Y 270.49,Z 463.051,A -85,B 0,C 180,E1 -18258.384,E2 -18258.384} C_VEL
LIN {X 0,Y 268.659,Z 474.655,A -85,B 0,C 180,E1 -18259.83,E2 -18259.83} C_VEL
LIN {X 0,Y 267.267,Z 485.011,A -85,B 0,C 180,E1 -18261.495,E2 -18261.495} C_VEL
LIN {X 0,Y 265.867,Z 493.512,A -85,B 0,C 180,E1 -18263.169,E2 -18263.169} C_VEL
LIN {X 0,Y 264.698,Z 501.331,A -85,B 0,C 180,E1 -18265.05,E2 -18265.05} C_VEL
LIN {X 0,Y 263.438,Z 508.988,A -85,B 0,C 180,E1 -18267.325,E2 -18267.325} C_VEL
LIN {X 0,Y 262.617,Z 514.232,A -85,B 0,C 180,E1 -18269.234,E2 -18269.234} C_VEL
LIN {X 0,Y 261.935,Z 519.31,A -85,B 0,C 180,E1 -18271.538,E2 -18271.538} C_VEL
LIN {X 0,Y 261.563,Z 523.256,A -85,B 0,C 180,E1 -18273.852,E2 -18273.852} C_VEL
LIN {X 0,Y 261.354,Z 526.178,A -85,B 0,C 180,E1 -18276.175,E2 -18276.175} C_VEL
LIN {X 0,Y 261.014,Z 528.575,A -85,B 0,C 180,E1 -18279.298,E2 -18279.298} C_VEL
LIN {X 0,Y 260.968,Z 529.187,A -85,B 0,C 180,E1 -18280.866,E2 -18280.866} C_VEL
LIN {X 0,Y 261.15,Z 529.38,A -85,B 0,C 180,E1 -18282.433,E2 -18282.433} C_VEL
LIN {X 0,Y 261.44,Z 528.973,A -85,B 0,C 180,E1 -18284.593,E2 -18284.593} C_VEL
LIN {X 0,Y 261.979,Z 527.5,A -85,B 0,C 180,E1 -18287.163,E2 -18287.163} C_VEL
LIN {X 0,Y 262.458,Z 526.023,A -85,B 0,C 180,E1 -18288.744,E2 -18288.744} C_VEL
LIN {X 0,Y 263.424,Z 523.193,A -85,B 0,C 180,E1 -18290.969,E2 -18290.969} C_VEL
LIN {X 0,Y 264.839,Z 518.826,A -85,B 0,C 180,E1 -18293.457,E2 -18293.457} C_VEL
LIN {X 0,Y 266.525,Z 513.442,A -85,B 0,C 180,E1 -18295.791,E2 -18295.791} C_VEL
LIN {X 0,Y 268.593,Z 506.643,A -85,B 0,C 180,E1 -18298.099,E2 -18298.099} C_VEL
LIN {X 0,Y 271.051,Z 498.138,A -85,B 0,C 180,E1 -18300.372,E2 -18300.372} C_VEL
LIN {X 0,Y 273.522,Z 488.906,A -85,B 0,C 180,E1 -18302.306,E2 -18302.306} C_VEL
LIN {X 0,Y 276.008,Z 478.348,A -85,B 0,C 180,E1 -18304.069,E2 -18304.069} C_VEL
LIN {X 0,Y 278.193,Z 467.307,A -85,B 0,C 180,E1 -18305.525,E2 -18305.525} C_VEL
LIN {X 0,Y 280.14,Z 455.327,A -85,B 0,C 180,E1 -18306.738,E2 -18306.738} C_VEL
LIN {X 0,Y 281.526,Z 444.229,A -85,B 0,C 180,E1 -18307.594,E2 -18307.594} C_VEL
LIN {X 0,Y 282.603,Z 431.067,A -85,B 0,C 180,E1 -18308.329,E2 -18308.329} C_VEL
LIN {X 0,Y 283.522,Z 416.574,A -85,B 0,C 180,E1 -18308.764,E2 -18308.764} C_VEL
LIN {X 0,Y 285.669,Z 362.568,A -85,B 0,C 180,E1 -18310.088,E2 -18310.088} C_VEL
LIN {X 0,Y 282.43,Z 354.576,A -85,B 0,C 180,E1 -18310.78,E2 -18310.78} C_VEL
LIN {X 0,Y 274.39,Z 338.296,A -85,B 0,C 180,E1 -18312.486,E2 -18312.486} C_VEL
LIN {X 0,Y 267.756,Z 326.655,A -85,B 0,C 180,E1 -18313.945,E2 -18313.945} C_VEL
LIN {X 0,Y 263.493,Z 319.229,A -85,B 0,C 180,E1 -18314.956,E2 -18314.956} C_VEL
LIN {X 0,Y 263.122,Z 317.71,A -85,B 0,C 180,E1 -18315.75,E2 -18315.75} C_VEL
LIN {X 0,Y 263.124,Z 317.709,A -85,B 0,C 180,E1 -18318.407,E2 -18318.407} C_VEL
LIN {X 0,Y 263.181,Z 317.696,A -85,B 0,C 180,E1 -18323.237,E2 -18323.237} C_VEL
LIN {X 0,Y 263.133,Z 317.7,A -85,B 0,C 180,E1 -18327.712,E2 -18327.712} C_VEL
LIN {X 0,Y 263.202,Z 317.688,A -85,B 0,C 180,E1 -18331.783,E2 -18331.783} C_VEL
LIN {X 0,Y 263.201,Z 317.692,A -85,B 0,C 180,E1 -18335.213,E2 -18335.213} C_VEL
LIN {X 0,Y 263.263,Z 317.682,A -85,B 0,C 180,E1 -18339.694,E2 -18339.694} C_VEL
LIN {X 0,Y 263.351,Z 317.671,A -85,B 0,C 180,E1 -18344.522,E2 -18344.522} C_VEL
LIN {X 0,Y 263.33,Z 317.678,A -85,B 0,C 180,E1 -18347.94,E2 -18347.94} C_VEL
LIN {X 0,Y 262.677,Z 317.756,A -85,B 0,C 180,E1 -18349.219,E2 -18349.219} C_VEL
LIN {X 0,Y 259.91,Z 318.109,A -85,B 0,C 180,E1 -18351.307,E2 -18351.307} C_VEL
LIN {X 0,Y 256.72,Z 318.497,A -85,B 0,C 180,E1 -18353.875,E2 -18353.875} C_VEL
LIN {X 0,Y 256.367,Z 318.543,A -85,B 0,C 180,E1 -18354.763,E2 -18354.763} C_VEL
LIN {X 0,Y 256.714,Z 318.497,A -85,B 0,C 180,E1 -18358.432,E2 -18358.432} C_VEL
LIN {X 0,Y 256.714,Z 318.5,A -85,B 0,C 180,E1 -18361.569,E2 -18361.569} C_VEL
LIN {X 0,Y 256.541,Z 318.516,A -85,B 0,C 180,E1 -18367.873,E2 -18367.873} C_VEL
LIN {X 0,Y 256.311,Z 318.546,A -85,B 0,C 180,E1 -18371.066,E2 -18371.066} C_VEL
LIN {X 0,Y 256.301,Z 318.547,A -85,B 0,C 180,E1 -18375.915,E2 -18375.915} C_VEL
LIN {X 0,Y 256.164,Z 318.566,A -85,B 0,C 180,E1 -18380.896,E2 -18380.896} C_VEL
LIN {X 0,Y 256.173,Z 318.567,A -85,B 0,C 180,E1 -18385.13,E2 -18385.13} C_VEL
LIN {X 0,Y 256.106,Z 318.579,A -85,B 0,C 180,E1 -18389.601,E2 -18389.601} C_VEL
LIN {X 0,Y 256.069,Z 318.583,A -85,B 0,C 180,E1 -18393.293,E2 -18393.293} C_VEL
LIN {X 0,Y 256.117,Z 318.58,A -85,B 0,C 180,E1 -18397.271,E2 -18397.271} C_VEL
LIN {X 0,Y 256.056,Z 318.563,A -85,B 0,C 180,E1 -18401.204,E2 -18401.204} C_VEL
LIN {X 0,Y 256.056,Z 318.591,A -85,B 0,C 180,E1 -18405.531,E2 -18405.531} C_VEL
LIN {X 0,Y 256.049,Z 318.594,A -85,B 0,C 180,E1 -18407.502,E2 -18407.502} C_VEL
LIN {X 0,Y 258.393,Z 326.703,A -85,B 0,C 180,E1 -18411.275,E2 -18411.275} C_VEL
LIN {X 0,Y 260.428,Z 334.6,A -85,B 0,C 180,E1 -18414.586,E2 -18414.586} C_VEL
LIN {X 0,Y 262.65,Z 338.795,A -85,B 0,C 180,E1 -18415.127,E2 -18415.127} C_VEL
LIN {X 0,Y 269.845,Z 353.134,A -85,B 0,C 180,E1 -18416.814,E2 -18416.814} C_VEL
LIN {X 0,Y 274.719,Z 364.227,A -85,B 0,C 180,E1 -18417.928,E2 -18417.928} C_VEL
LIN {X 0,Y 278.317,Z 384.884,A -85,B 0,C 180,E1 -18419.101,E2 -18419.101} C_VEL
LIN {X 0,Y 278.839,Z 389.542,A -85,B 0,C 180,E1 -18419.319,E2 -18419.319} C_VEL
LIN {X 0,Y 276.587,Z 444.419,A -85,B 0,C 180,E1 -18420.741,E2 -18420.741} C_VEL
LIN {X 0,Y 275.324,Z 457.75,A -85,B 0,C 180,E1 -18421.353,E2 -18421.353} C_VEL
LIN {X 0,Y 273.459,Z 470.723,A -85,B 0,C 180,E1 -18422.236,E2 -18422.236} C_VEL
LIN {X 0,Y 271.127,Z 483.275,A -85,B 0,C 180,E1 -18423.439,E2 -18423.439} C_VEL
LIN {X 0,Y 268.626,Z 494.472,A -85,B 0,C 180,E1 -18424.84,E2 -18424.84} C_VEL
LIN {X 0,Y 266.135,Z 504.579,A -85,B 0,C 180,E1 -18426.458,E2 -18426.458} C_VEL
LIN {X 0,Y 263.344,Z 514.518,A -85,B 0,C 180,E1 -18428.472,E2 -18428.472} C_VEL
LIN {X 0,Y 261.091,Z 522.186,A -85,B 0,C 180,E1 -18430.412,E2 -18430.412} C_VEL
LIN {X 0,Y 259.097,Z 529.251,A -85,B 0,C 180,E1 -18432.64,E2 -18432.64} C_VEL
LIN {X 0,Y 257.272,Z 535.139,A -85,B 0,C 180,E1 -18434.958,E2 -18434.958} C_VEL
LIN {X 0,Y 255.818,Z 539.802,A -85,B 0,C 180,E1 -18437.303,E2 -18437.303} C_VEL
LIN {X 0,Y 254.919,Z 543.379,A -85,B 0,C 180,E1 -18439.676,E2 -18439.676} C_VEL
LIN {X 0,Y 254.314,Z 545.968,A -85,B 0,C 180,E1 -18442.057,E2 -18442.057} C_VEL
LIN {X 0,Y 253.985,Z 547.909,A -85,B 0,C 180,E1 -18444.978,E2 -18444.978} C_VEL
LIN {X 0,Y 254.02,Z 548.407,A -85,B 0,C 180,E1 -18446.827,E2 -18446.827} C_VEL
LIN {X 0,Y 254.068,Z 548.426,A -85,B 0,C 180,E1 -18448.414,E2 -18448.414} C_VEL
LIN {X 0,Y 254.101,Z 548.059,A -85,B 0,C 180,E1 -18449.999,E2 -18449.999} C_VEL
LIN {X 0,Y 254.092,Z 547.267,A -85,B 0,C 180,E1 -18451.584,E2 -18451.584} C_VEL
LIN {X 0,Y 254.063,Z 546.042,A -85,B 0,C 180,E1 -18453.171,E2 -18453.171} C_VEL
LIN {X 0,Y 254.087,Z 543.799,A -85,B 0,C 180,E1 -18455.277,E2 -18455.277} C_VEL
LIN {X 0,Y 254.304,Z 539.768,A -85,B 0,C 180,E1 -18457.942,E2 -18457.942} C_VEL
LIN {X 0,Y 254.733,Z 534.976,A -85,B 0,C 180,E1 -18460.33,E2 -18460.33} C_VEL
LIN {X 0,Y 255.684,Z 527.777,A -85,B 0,C 180,E1 -18463.106,E2 -18463.106} C_VEL
LIN {X 0,Y 256.921,Z 519.915,A -85,B 0,C 180,E1 -18465.468,E2 -18465.468} C_VEL
LIN {X 0,Y 258.306,Z 511.876,A -85,B 0,C 180,E1 -18467.414,E2 -18467.414} C_VEL
LIN {X 0,Y 259.691,Z 502.022,A -85,B 0,C 180,E1 -18469.36,E2 -18469.36} C_VEL
LIN {X 0,Y 261.43,Z 491.084,A -85,B 0,C 180,E1 -18471.072,E2 -18471.072} C_VEL
LIN {X 0,Y 262.957,Z 480.367,A -85,B 0,C 180,E1 -18472.386,E2 -18472.386} C_VEL
LIN {X 0,Y 264.473,Z 467.438,A -85,B 0,C 180,E1 -18473.594,E2 -18473.594} C_VEL
LIN {X 0,Y 265.702,Z 454.345,A -85,B 0,C 180,E1 -18474.463,E2 -18474.463} C_VEL
LIN {X 0,Y 266.46,Z 440.814,A -85,B 0,C 180,E1 -18475.027,E2 -18475.027} C_VEL
LIN {X 0,Y 267.967,Z 384.831,A -85,B 0,C 180,E1 -18476.506,E2 -18476.506} C_VEL
LIN {X 0,Y 263.536,Z 349.106,A -85,B 0,C 180,E1 -18477.946,E2 -18477.946} C_VEL
LIN {X 0,Y 262.36,Z 342.983,A -85,B 0,C 180,E1 -18478.24,E2 -18478.24} C_VEL
LIN {X 0,Y 259.734,Z 335.552,A -85,B 0,C 180,E1 -18478.734,E2 -18478.734} C_VEL
LIN {X 0,Y 257.477,Z 324.694,A -85,B 0,C 180,E1 -18482.559,E2 -18482.559} C_VEL
LIN {X 0,Y 256.113,Z 318.583,A -85,B 0,C 180,E1 -18484.819,E2 -18484.819} C_VEL
LIN {X 0,Y 256.121,Z 318.58,A -85,B 0,C 180,E1 -18487.272,E2 -18487.272} C_VEL
LIN {X 0,Y 256.053,Z 318.589,A -85,B 0,C 180,E1 -18491.202,E2 -18491.202} C_VEL
LIN {X 0,Y 256.039,Z 318.59,A -85,B 0,C 180,E1 -18495.533,E2 -18495.533} C_VEL
LIN {X 0,Y 256.053,Z 318.592,A -85,B 0,C 180,E1 -18498.796,E2 -18498.796} C_VEL
LIN {X 0,Y 256.128,Z 318.584,A -85,B 0,C 180,E1 -18502.866,E2 -18502.866} C_VEL
LIN {X 0,Y 256.065,Z 318.592,A -85,B 0,C 180,E1 -18506.706,E2 -18506.706} C_VEL
LIN {X 0,Y 256.111,Z 318.584,A -85,B 0,C 180,E1 -18510.4,E2 -18510.4} C_VEL
LIN {X 0,Y 256.185,Z 318.574,A -85,B 0,C 180,E1 -18514.861,E2 -18514.861} C_VEL
LIN {X 0,Y 256.164,Z 318.577,A -85,B 0,C 180,E1 -18519.104,E2 -18519.104} C_VEL
LIN {X 0,Y 256.297,Z 318.557,A -85,B 0,C 180,E1 -18524.084,E2 -18524.084} C_VEL
LIN {X 0,Y 256.306,Z 318.544,A -85,B 0,C 180,E1 -18528.933,E2 -18528.933} C_VEL
LIN {X 0,Y 256.534,Z 318.527,A -85,B 0,C 180,E1 -18532.127,E2 -18532.127} C_VEL
LIN {X 0,Y 256.71,Z 318.494,A -85,B 0,C 180,E1 -18538.431,E2 -18538.431} C_VEL
LIN {X 0,Y 256.709,Z 318.501,A -85,B 0,C 180,E1 -18541.568,E2 -18541.568} C_VEL
LIN {X 0,Y 256.451,Z 318.534,A -85,B 0,C 180,E1 -18546.568,E2 -18546.568} C_VEL
LIN {X 0,Y 256.423,Z 318.531,A -85,B 0,C 180,E1 -18549.465,E2 -18549.465} C_VEL
LIN {X 0,Y 256.251,Z 318.566,A -85,B 0,C 180,E1 -18554.29,E2 -18554.29} C_VEL
LIN {X 0,Y 256.205,Z 318.567,A -85,B 0,C 180,E1 -18557.562,E2 -18557.562} C_VEL
LIN {X 0,Y 256.149,Z 318.566,A -85,B 0,C 180,E1 -18561.117,E2 -18561.117} C_VEL
LIN {X 0,Y 256.167,Z 318.574,A -85,B 0,C 180,E1 -18565.13,E2 -18565.13} C_VEL
LIN {X 0,Y 256.11,Z 318.57,A -85,B 0,C 180,E1 -18569.6,E2 -18569.6} C_VEL
LIN {X 0,Y 256.064,Z 318.585,A -85,B 0,C 180,E1 -18573.293,E2 -18573.293} C_VEL
LIN {X 0,Y 256.109,Z 318.574,A -85,B 0,C 180,E1 -18577.271,E2 -18577.271} C_VEL
LIN {X 0,Y 256.051,Z 318.589,A -85,B 0,C 180,E1 -18581.204,E2 -18581.204} C_VEL
LIN {X 0,Y 256.022,Z 318.584,A -85,B 0,C 180,E1 -18585.538,E2 -18585.538} C_VEL
LIN {X 0,Y 256.015,Z 318.594,A -85,B 0,C 180,E1 -18588.79,E2 -18588.79} C_VEL
LIN {X 0,Y 256.125,Z 318.577,A -85,B 0,C 180,E1 -18592.868,E2 -18592.868} C_VEL
LIN {X 0,Y 256.062,Z 318.588,A -85,B 0,C 180,E1 -18596.707,E2 -18596.707} C_VEL
LIN {X 0,Y 256.038,Z 318.586,A -85,B 0,C 180,E1 -18600.392,E2 -18600.392} C_VEL
LIN {X 0,Y 256.069,Z 318.586,A -85,B 0,C 180,E1 -18603.952,E2 -18603.952} C_VEL
LIN {X 0,Y 256.07,Z 318.589,A -85,B 0,C 180,E1 -18607.404,E2 -18607.404} C_VEL
LIN {X 0,Y 256.198,Z 318.717,A -85,B 0,C 180,E1 -18610.999,E2 -18610.999} C_VEL
LIN {X 0,Y 257.356,Z 321.676,A -85,B 0,C 180,E1 -18611.211,E2 -18611.211} C_VEL
LIN {X 0,Y 263.42,Z 336.327,A -85,B 0,C 180,E1 -18612.258,E2 -18612.258} C_VEL
LIN {X 0,Y 268.595,Z 351.192,A -85,B 0,C 180,E1 -18613.178,E2 -18613.178} C_VEL
LIN {X 0,Y 268.724,Z 356.295,A -85,B 0,C 180,E1 -18613.336,E2 -18613.336} C_VEL
LIN {X 0,Y 266.675,Z 426.486,A -85,B 0,C 180,E1 -18615.209,E2 -18615.209} C_VEL
LIN {X 0,Y 265.91,Z 440.158,A -85,B 0,C 180,E1 -18615.899,E2 -18615.899} C_VEL
LIN {X 0,Y 264.862,Z 452.976,A -85,B 0,C 180,E1 -18616.868,E2 -18616.868} C_VEL
LIN {X 0,Y 263.613,Z 464.669,A -85,B 0,C 180,E1 -18618.076,E2 -18618.076} C_VEL
LIN {X 0,Y 261.901,Z 474.744,A -85,B 0,C 180,E1 -18619.369,E2 -18619.369} C_VEL
LIN {X 0,Y 260.439,Z 485.132,A -85,B 0,C 180,E1 -18621.074,E2 -18621.074} C_VEL
LIN {X 0,Y 258.848,Z 494.524,A -85,B 0,C 180,E1 -18622.983,E2 -18622.983} C_VEL
LIN {X 0,Y 257.393,Z 503.554,A -85,B 0,C 180,E1 -18625.302,E2 -18625.302} C_VEL
LIN {X 0,Y 256.118,Z 510.853,A -85,B 0,C 180,E1 -18627.642,E2 -18627.642} C_VEL
LIN {X 0,Y 255.29,Z 516.694,A -85,B 0,C 180,E1 -18630.001,E2 -18630.001} C_VEL
LIN {X 0,Y 254.618,Z 521.312,A -85,B 0,C 180,E1 -18632.373,E2 -18632.373} C_VEL
LIN {X 0,Y 254.382,Z 524.82,A -85,B 0,C 180,E1 -18634.755,E2 -18634.755} C_VEL
LIN {X 0,Y 254.233,Z 526.605,A -85,B 0,C 180,E1 -18636.349,E2 -18636.349} C_VEL
LIN {X 0,Y 254.008,Z 527.966,A -85,B 0,C 180,E1 -18637.952,E2 -18637.952} C_VEL
LIN {X 0,Y 253.897,Z 528.931,A -85,B 0,C 180,E1 -18639.561,E2 -18639.561} C_VEL
LIN {X 0,Y 253.894,Z 529.503,A -85,B 0,C 180,E1 -18641.173,E2 -18641.173} C_VEL
LIN {X 0,Y 254.085,Z 529.631,A -85,B 0,C 180,E1 -18642.785,E2 -18642.785} C_VEL
LIN {X 0,Y 254.389,Z 529.255,A -85,B 0,C 180,E1 -18644.774,E2 -18644.774} C_VEL
LIN {X 0,Y 255.02,Z 527.633,A -85,B 0,C 180,E1 -18647.647,E2 -18647.647} C_VEL
LIN {X 0,Y 255.574,Z 526.095,A -85,B 0,C 180,E1 -18649.268,E2 -18649.268} C_VEL
LIN {X 0,Y 256.484,Z 523.562,A -85,B 0,C 180,E1 -18651.308,E2 -18651.308} C_VEL
LIN {X 0,Y 258.153,Z 518.737,A -85,B 0,C 180,E1 -18654.102,E2 -18654.102} C_VEL
LIN {X 0,Y 259.838,Z 513.566,A -85,B 0,C 180,E1 -18656.378,E2 -18656.378} C_VEL
LIN {X 0,Y 262.166,Z 506.364,A -85,B 0,C 180,E1 -18658.851,E2 -18658.851} C_VEL
LIN {X 0,Y 264.308,Z 499.276,A -85,B 0,C 180,E1 -18660.788,E2 -18660.788} C_VEL
LIN {X 0,Y 266.819,Z 490.476,A -85,B 0,C 180,E1 -18662.731,E2 -18662.731} C_VEL
LIN {X 0,Y 269.438,Z 479.981,A -85,B 0,C 180,E1 -18664.564,E2 -18664.564} C_VEL
LIN {X 0,Y 271.678,Z 469.292,A -85,B 0,C 180,E1 -18666.052,E2 -18666.052} C_VEL
LIN {X 0,Y 273.782,Z 457.632,A -85,B 0,C 180,E1 -18667.308,E2 -18667.308} C_VEL
LIN {X 0,Y 275.458,Z 444.886,A -85,B 0,C 180,E1 -18668.339,E2 -18668.339} C_VEL
LIN {X 0,Y 276.595,Z 431.925,A -85,B 0,C 180,E1 -18669.084,E2 -18669.084} C_VEL
LIN {X 0,Y 277.499,Z 418.843,A -85,B 0,C 180,E1 -18669.505,E2 -18669.505} C_VEL
LIN {X 0,Y 279.768,Z 364.205,A -85,B 0,C 180,E1 -18670.865,E2 -18670.865} C_VEL
LIN {X 0,Y 272.919,Z 349.106,A -85,B 0,C 180,E1 -18672.367,E2 -18672.367} C_VEL
LIN {X 0,Y 265.559,Z 335.347,A -85,B 0,C 180,E1 -18674.024,E2 -18674.024} C_VEL
LIN {X 0,Y 258.551,Z 323.491,A -85,B 0,C 180,E1 -18675.686,E2 -18675.686} C_VEL
LIN {X 0,Y 256.484,Z 320.257,A -85,B 0,C 180,E1 -18676.193,E2 -18676.193} C_VEL
LIN {X 0,Y 256.23,Z 319.476,A -85,B 0,C 180,E1 -18676.329,E2 -18676.329} C_VEL
LIN {X 0,Y 256.044,Z 318.592,A -85,B 0,C 180,E1 -18676.83,E2 -18676.83} C_VEL
LIN {X 0,Y 256.071,Z 318.585,A -85,B 0,C 180,E1 -18680.858,E2 -18680.858} C_VEL
LIN {X 0,Y 256.13,Z 318.576,A -85,B 0,C 180,E1 -18682.868,E2 -18682.868} C_VEL
LIN {X 0,Y 256.068,Z 318.58,A -85,B 0,C 180,E1 -18686.708,E2 -18686.708} C_VEL
LIN {X 0,Y 256.114,Z 318.573,A -85,B 0,C 180,E1 -18690.401,E2 -18690.401} C_VEL
LIN {X 0,Y 256.171,Z 318.57,A -85,B 0,C 180,E1 -18694.87,E2 -18694.87} C_VEL
LIN {X 0,Y 256.163,Z 318.572,A -85,B 0,C 180,E1 -18699.105,E2 -18699.105} C_VEL
LIN {X 0,Y 256.3,Z 318.551,A -85,B 0,C 180,E1 -18704.085,E2 -18704.085} C_VEL
LIN {X 0,Y 256.31,Z 318.548,A -85,B 0,C 180,E1 -18708.934,E2 -18708.934} C_VEL
LIN {X 0,Y 256.541,Z 318.525,A -85,B 0,C 180,E1 -18712.127,E2 -18712.127} C_VEL
LIN {X 0,Y 256.367,Z 318.543,A -85,B 0,C 180,E1 -18714.763,E2 -18714.763} C_VEL
LIN {X 0,Y 255.716,Z 318.633,A -85,B 0,C 180,E1 -18716.076,E2 -18716.076} C_VEL
LIN {X 0,Y 253.129,Z 318.96,A -85,B 0,C 180,E1 -18718.228,E2 -18718.228} C_VEL
LIN {X 0,Y 250.067,Z 319.332,A -85,B 0,C 180,E1 -18720.868,E2 -18720.868} C_VEL
LIN {X 0,Y 249.643,Z 319.378,A -85,B 0,C 180,E1 -18721.777,E2 -18721.777} C_VEL
LIN {X 0,Y 249.462,Z 319.398,A -85,B 0,C 180,E1 -18726.471,E2 -18726.471} C_VEL
LIN {X 0,Y 249.39,Z 319.417,A -85,B 0,C 180,E1 -18729.735,E2 -18729.735} C_VEL
LIN {X 0,Y 249.207,Z 319.437,A -85,B 0,C 180,E1 -18734.704,E2 -18734.704} C_VEL
LIN {X 0,Y 249.141,Z 319.448,A -85,B 0,C 180,E1 -18738.078,E2 -18738.078} C_VEL
LIN {X 0,Y 249.086,Z 319.452,A -85,B 0,C 180,E1 -18741.519,E2 -18741.519} C_VEL
LIN {X 0,Y 249.119,Z 319.447,A -85,B 0,C 180,E1 -18745.476,E2 -18745.476} C_VEL
LIN {X 0,Y 249.076,Z 319.451,A -85,B 0,C 180,E1 -18748.99,E2 -18748.99} C_VEL
LIN {X 0,Y 249.032,Z 319.456,A -85,B 0,C 180,E1 -18752.426,E2 -18752.426} C_VEL
LIN {X 0,Y 249.032,Z 319.456,A -85,B 0,C 180,E1 -18756.346,E2 -18756.346} C_VEL
LIN {X 0,Y 248.993,Z 319.44,A -85,B 0,C 180,E1 -18760.481,E2 -18760.481} C_VEL
LIN {X 0,Y 249.003,Z 319.464,A -85,B 0,C 180,E1 -18762.791,E2 -18762.791} C_VEL
LIN {X 0,Y 249.032,Z 319.557,A -85,B 0,C 180,E1 -18766.358,E2 -18766.358} C_VEL
LIN {X 0,Y 251.431,Z 327.856,A -85,B 0,C 180,E1 -18770.406,E2 -18770.406} C_VEL
LIN {X 0,Y 253.186,Z 334.315,A -85,B 0,C 180,E1 -18773.22,E2 -18773.22} C_VEL
LIN {X 0,Y 255.552,Z 338.679,A -85,B 0,C 180,E1 -18773.834,E2 -18773.834} C_VEL
LIN {X 0,Y 263.214,Z 353.659,A -85,B 0,C 180,E1 -18775.735,E2 -18775.735} C_VEL
LIN {X 0,Y 269.251,Z 367.049,A -85,B 0,C 180,E1 -18777.175,E2 -18777.175} C_VEL
LIN {X 0,Y 272.809,Z 388.152,A -85,B 0,C 180,E1 -18778.402,E2 -18778.402} C_VEL
LIN {X 0,Y 272.904,Z 392.232,A -85,B 0,C 180,E1 -18778.545,E2 -18778.545} C_VEL
LIN {X 0,Y 270.676,Z 443.976,A -85,B 0,C 180,E1 -18779.907,E2 -18779.907} C_VEL
LIN {X 0,Y 269.349,Z 457.683,A -85,B 0,C 180,E1 -18780.549,E2 -18780.549} C_VEL
LIN {X 0,Y 267.415,Z 470.591,A -85,B 0,C 180,E1 -18781.445,E2 -18781.445} C_VEL
LIN {X 0,Y 265.179,Z 482.325,A -85,B 0,C 180,E1 -18782.581,E2 -18782.581} C_VEL
LIN {X 0,Y 262.56,Z 493.647,A -85,B 0,C 180,E1 -18784.003,E2 -18784.003} C_VEL
LIN {X 0,Y 259.944,Z 503.874,A -85,B 0,C 180,E1 -18785.65,E2 -18785.65} C_VEL
